KUKA KRL data list: CNC4.dat

&ACCESS RV
DEFDAT CNC4 Public
DECL GLOBAL FRAME gfCNCPoint4[30000]


gfCNCPoint4[1] = {X 250.4410, Y 22.5668, Z -3.9870, A 0.000, B 0.000, C 0.000 }
gfCNCPoint4[2] = {X 251.6873, Y 22.5560, Z -4.3210, A 0.000, B 0.000, C 0.000 }
gfCNCPoint4[3] = {X 252.9774, Y 22.5560, Z -4.6667, A 0.000, B 0.000, C 0.000 }
gfCNCPoint4[4] = {X 257.4115, Y 22.5560, Z -4.6667, A 0.000, B 0.000, C 0.000 }
gfCNCPoint4[5] = {X 257.4115, Y 19.7811, Z -4.6667, A 0.000, B 0.000, C 0.000 }
gfCNCPoint4[6] = {X 251.5292, Y 19.7811, Z -4.6667, A 0.000, B 0.000, C 0.000 }
gfCNCPoint4[7] = {X 250.8345, Y 19.7919, Z -4.6667, A 0.000, B 0.000, C 0.000 }
gfCNCPoint4[8] = {X 249.8296, Y 19.8652, Z -4.6667, A 0.000, B 0.000, C 0.000 }
gfCNCPoint4[9] = {X 248.8453, Y 20.0800, Z -4.6667, A 0.000, B 0.000, C 0.000 }
gfCNCPoint4[10] = {X 248.7005, Y 20.1571, Z -4.6667, A 0.000, B 0.000, C 0.000 }
gfCNCPoint4[11] = {X 248.6143, Y 20.2967, Z -4.6667, A 0.000, B 0.000, C 0.000 }
gfCNCPoint4[12] = {X 248.4764, Y 20.9719, Z -4.6667, A 0.000, B 0.000, C 0.000 }
gfCNCPoint4[13] = {X 248.4575, Y 21.6608, Z -4.6667, A 0.000, B 0.000, C 0.000 }
gfCNCPoint4[14] = {X 248.5584, Y 22.3425, Z -4.6667, A 0.000, B 0.000, C 0.000 }
gfCNCPoint4[15] = {X 248.8771, Y 22.4203, Z -4.6667, A 0.000, B 0.000, C 0.000 }
gfCNCPoint4[16] = {X 249.2022, Y 22.4644, Z -4.6667, A 0.000, B 0.000, C 0.000 }
gfCNCPoint4[17] = {X 250.4437, Y 22.5386, Z -4.6667, A 0.000, B 0.000, C 0.000 }
gfCNCPoint4[18] = {X 251.6873, Y 22.5560, Z -4.6667, A 0.000, B 0.000, C 0.000 }
gfCNCPoint4[19] = {X 252.9774, Y 22.5560, Z -4.6667, A 0.000, B 0.000, C 0.000 }
gfCNCPoint4[20] = {X 248.9926, Y 22.2874, Z -4.6667, A 0.000, B 0.000, C 0.000 }
gfCNCPoint4[21] = {X 252.9774, Y 22.6360, Z -4.6667, A 0.000, B 0.000, C 0.000 }
gfCNCPoint4[22] = {X 257.4915, Y 22.6360, Z -4.6667, A 0.000, B 0.000, C 0.000 }
gfCNCPoint4[23] = {X 257.4915, Y 19.7011, Z -4.6667, A 0.000, B 0.000, C 0.000 }
gfCNCPoint4[24] = {X 251.5286, Y 19.7011, Z -4.6667, A 0.000, B 0.000, C 0.000 }
gfCNCPoint4[25] = {X 250.8365, Y 19.7119, Z -4.6667, A 0.000, B 0.000, C 0.000 }
gfCNCPoint4[26] = {X 249.8259, Y 19.7853, Z -4.6667, A 0.000, B 0.000, C 0.000 }
gfCNCPoint4[27] = {X 248.8356, Y 20.0002, Z -4.6667, A 0.000, B 0.000, C 0.000 }
gfCNCPoint4[28] = {X 248.6488, Y 20.0958, Z -4.6667, A 0.000, B 0.000, C 0.000 }
gfCNCPoint4[29] = {X 248.5376, Y 20.2739, Z -4.6667, A 0.000, B 0.000, C 0.000 }
gfCNCPoint4[30] = {X 248.3952, Y 20.9779, Z -4.6667, A 0.000, B 0.000, C 0.000 }
gfCNCPoint4[31] = {X 248.3796, Y 21.6960, Z -4.6667, A 0.000, B 0.000, C 0.000 }
gfCNCPoint4[32] = {X 248.4915, Y 22.4056, Z -4.6667, A 0.000, B 0.000, C 0.000 }
gfCNCPoint4[33] = {X 248.8397, Y 22.4946, Z -4.6667, A 0.000, B 0.000, C 0.000 }
gfCNCPoint4[34] = {X 249.1956, Y 22.5442, Z -4.6667, A 0.000, B 0.000, C 0.000 }
gfCNCPoint4[35] = {X 250.4397, Y 22.6185, Z -4.6667, A 0.000, B 0.000, C 0.000 }
gfCNCPoint4[36] = {X 251.6859, Y 22.6360, Z -4.6667, A 0.000, B 0.000, C 0.000 }
gfCNCPoint4[37] = {X 252.9774, Y 22.6360, Z -4.6667, A 0.000, B 0.000, C 0.000 }
gfCNCPoint4[38] = {X 256.9621, Y 22.2874, Z -4.6667, A 0.000, B 0.000, C 0.000 }
gfCNCPoint4[39] = {X 248.9926, Y 22.3674, Z -4.6667, A 0.000, B 0.000, C 0.000 }
gfCNCPoint4[40] = {X 252.9774, Y 22.7160, Z -4.6667, A 0.000, B 0.000, C 0.000 }
gfCNCPoint4[41] = {X 257.5715, Y 22.7160, Z -4.6667, A 0.000, B 0.000, C 0.000 }
gfCNCPoint4[42] = {X 257.5715, Y 19.6211, Z -4.6667, A 0.000, B 0.000, C 0.000 }
gfCNCPoint4[43] = {X 251.5280, Y 19.6211, Z -4.6667, A 0.000, B 0.000, C 0.000 }
gfCNCPoint4[44] = {X 250.8358, Y 19.6319, Z -4.6667, A 0.000, B 0.000, C 0.000 }
gfCNCPoint4[45] = {X 249.8156, Y 19.7059, Z -4.6667, A 0.000, B 0.000, C 0.000 }
gfCNCPoint4[46] = {X 248.8160, Y 19.9226, Z -4.6667, A 0.000, B 0.000, C 0.000 }
gfCNCPoint4[47] = {X 248.5934, Y 20.0381, Z -4.6667, A 0.000, B 0.000, C 0.000 }
gfCNCPoint4[48] = {X 248.4609, Y 20.2511, Z -4.6667, A 0.000, B 0.000, C 0.000 }
gfCNCPoint4[49] = {X 248.3140, Y 20.9838, Z -4.6667, A 0.000, B 0.000, C 0.000 }
gfCNCPoint4[50] = {X 248.3019, Y 21.7310, Z -4.6667, A 0.000, B 0.000, C 0.000 }
gfCNCPoint4[51] = {X 248.4249, Y 22.4681, Z -4.6667, A 0.000, B 0.000, C 0.000 }
gfCNCPoint4[52] = {X 248.8023, Y 22.5687, Z -4.6667, A 0.000, B 0.000, C 0.000 }
gfCNCPoint4[53] = {X 249.1890, Y 22.6239, Z -4.6667, A 0.000, B 0.000, C 0.000 }
gfCNCPoint4[54] = {X 250.4366, Y 22.6984, Z -4.6667, A 0.000, B 0.000, C 0.000 }
gfCNCPoint4[55] = {X 251.6863, Y 22.7160, Z -4.6667, A 0.000, B 0.000, C 0.000 }
gfCNCPoint4[56] = {X 252.9774, Y 22.7160, Z -4.6667, A 0.000, B 0.000, C 0.000 }
gfCNCPoint4[57] = {X 256.9621, Y 22.3674, Z -4.6667, A 0.000, B 0.000, C 0.000 }
gfCNCPoint4[58] = {X 248.9926, Y 22.4474, Z -4.6667, A 0.000, B 0.000, C 0.000 }
gfCNCPoint4[59] = {X 252.9774, Y 22.7960, Z -4.6667, A 0.000, B 0.000, C 0.000 }
gfCNCPoint4[60] = {X 257.6515, Y 22.7960, Z -4.6667, A 0.000, B 0.000, C 0.000 }
gfCNCPoint4[61] = {X 257.6515, Y 19.5411, Z -4.6667, A 0.000, B 0.000, C 0.000 }
gfCNCPoint4[62] = {X 251.5274, Y 19.5411, Z -4.6667, A 0.000, B 0.000, C 0.000 }
gfCNCPoint4[63] = {X 250.8351, Y 19.5519, Z -4.6667, A 0.000, B 0.000, C 0.000 }
gfCNCPoint4[64] = {X 249.8053, Y 19.6266, Z -4.6667, A 0.000, B 0.000, C 0.000 }
gfCNCPoint4[65] = {X 248.7962, Y 19.8450, Z -4.6667, A 0.000, B 0.000, C 0.000 }
gfCNCPoint4[66] = {X 248.5379, Y 19.9805, Z -4.6667, A 0.000, B 0.000, C 0.000 }
gfCNCPoint4[67] = {X 248.3842, Y 20.2283, Z -4.6667, A 0.000, B 0.000, C 0.000 }
gfCNCPoint4[68] = {X 248.2330, Y 20.9896, Z -4.6667, A 0.000, B 0.000, C 0.000 }
gfCNCPoint4[69] = {X 248.2244, Y 21.7657, Z -4.6667, A 0.000, B 0.000, C 0.000 }
gfCNCPoint4[70] = {X 248.3587, Y 22.5302, Z -4.6667, A 0.000, B 0.000, C 0.000 }
gfCNCPoint4[71] = {X 248.7651, Y 22.6427, Z -4.6667, A 0.000, B 0.000, C 0.000 }
gfCNCPoint4[72] = {X 249.1825, Y 22.7036, Z -4.6667, A 0.000, B 0.000, C 0.000 }
gfCNCPoint4[73] = {X 250.4335, Y 22.7784, Z -4.6667, A 0.000, B 0.000, C 0.000 }
gfCNCPoint4[74] = {X 251.6866, Y 22.7960, Z -4.6667, A 0.000, B 0.000, C 0.000 }
gfCNCPoint4[75] = {X 252.9774, Y 22.7960, Z -4.6667, A 0.000, B 0.000, C 0.000 }
gfCNCPoint4[76] = {X 256.9621, Y 22.4474, Z -4.6667, A 0.000, B 0.000, C 0.000 }
gfCNCPoint4[77] = {X 248.9926, Y 22.5274, Z -4.6667, A 0.000, B 0.000, C 0.000 }
gfCNCPoint4[78] = {X 252.9774, Y 22.8760, Z -4.6667, A 0.000, B 0.000, C 0.000 }
gfCNCPoint4[79] = {X 257.7315, Y 22.8760, Z -4.6667, A 0.000, B 0.000, C 0.000 }
gfCNCPoint4[80] = {X 257.7315, Y 19.4611, Z -4.6667, A 0.000, B 0.000, C 0.000 }
gfCNCPoint4[81] = {X 251.5267, Y 19.4611, Z -4.6667, A 0.000, B 0.000, C 0.000 }
gfCNCPoint4[82] = {X 250.8343, Y 19.4719, Z -4.6667, A 0.000, B 0.000, C 0.000 }
gfCNCPoint4[83] = {X 249.7949, Y 19.5472, Z -4.6667, A 0.000, B 0.000, C 0.000 }
gfCNCPoint4[84] = {X 248.7763, Y 19.7675, Z -4.6667, A 0.000, B 0.000, C 0.000 }
gfCNCPoint4[85] = {X 248.4824, Y 19.9229, Z -4.6667, A 0.000, B 0.000, C 0.000 }
gfCNCPoint4[86] = {X 248.3075, Y 20.2056, Z -4.6667, A 0.000, B 0.000, C 0.000 }
gfCNCPoint4[87] = {X 248.1526, Y 20.9889, Z -4.6667, A 0.000, B 0.000, C 0.000 }
gfCNCPoint4[88] = {X 248.1459, Y 21.7874, Z -4.6667, A 0.000, B 0.000, C 0.000 }
gfCNCPoint4[89] = {X 248.2876, Y 22.5732, Z -4.6667, A 0.000, B 0.000, C 0.000 }
gfCNCPoint4[90] = {X 248.3062, Y 22.5966, Z -4.6667, A 0.000, B 0.000, C 0.000 }
gfCNCPoint4[91] = {X 248.3326, Y 22.6058, Z -4.6667, A 0.000, B 0.000, C 0.000 }
gfCNCPoint4[92] = {X 248.7487, Y 22.7210, Z -4.6667, A 0.000, B 0.000, C 0.000 }
gfCNCPoint4[93] = {X 249.1759, Y 22.7833, Z -4.6667, A 0.000, B 0.000, C 0.000 }
gfCNCPoint4[94] = {X 250.4304, Y 22.8583, Z -4.6667, A 0.000, B 0.000, C 0.000 }
gfCNCPoint4[95] = {X 251.6870, Y 22.8760, Z -4.6667, A 0.000, B 0.000, C 0.000 }
gfCNCPoint4[96] = {X 252.9774, Y 22.8760, Z -4.6667, A 0.000, B 0.000, C 0.000 }
gfCNCPoint4[97] = {X 256.9621, Y 22.5274, Z -4.6667, A 0.000, B 0.000, C 0.000 }
gfCNCPoint4[98] = {X 248.9926, Y 22.6074, Z -4.6667, A 0.000, B 0.000, C 0.000 }
gfCNCPoint4[99] = {X 252.9774, Y 22.9560, Z -4.6667, A 0.000, B 0.000, C 0.000 }
gfCNCPoint4[100] = {X 257.8115, Y 22.9560, Z -4.6667, A 0.000, B 0.000, C 0.000 }
gfCNCPoint4[101] = {X 257.8115, Y 19.3811, Z -4.6667, A 0.000, B 0.000, C 0.000 }
gfCNCPoint4[102] = {X 251.5261, Y 19.3811, Z -4.6667, A 0.000, B 0.000, C 0.000 }
gfCNCPoint4[103] = {X 250.8336, Y 19.3919, Z -4.6667, A 0.000, B 0.000, C 0.000 }
gfCNCPoint4[104] = {X 249.7844, Y 19.4679, Z -4.6667, A 0.000, B 0.000, C 0.000 }
gfCNCPoint4[105] = {X 248.7562, Y 19.6901, Z -4.6667, A 0.000, B 0.000, C 0.000 }
gfCNCPoint4[106] = {X 248.4268, Y 19.8653, Z -4.6667, A 0.000, B 0.000, C 0.000 }
gfCNCPoint4[107] = {X 248.2308, Y 20.1828, Z -4.6667, A 0.000, B 0.000, C 0.000 }
gfCNCPoint4[108] = {X 248.0725, Y 20.9862, Z -4.6667, A 0.000, B 0.000, C 0.000 }
gfCNCPoint4[109] = {X 248.0671, Y 21.8050, Z -4.6667, A 0.000, B 0.000, C 0.000 }
gfCNCPoint4[110] = {X 248.2149, Y 22.6104, Z -4.6667, A 0.000, B 0.000, C 0.000 }
gfCNCPoint4[111] = {X 248.2579, Y 22.6642, Z -4.6667, A 0.000, B 0.000, C 0.000 }
gfCNCPoint4[112] = {X 248.7070, Y 22.7939, Z -4.6667, A 0.000, B 0.000, C 0.000 }
gfCNCPoint4[113] = {X 249.1693, Y 22.8631, Z -4.6667, A 0.000, B 0.000, C 0.000 }
gfCNCPoint4[114] = {X 250.4273, Y 22.9382, Z -4.6667, A 0.000, B 0.000, C 0.000 }
gfCNCPoint4[115] = {X 251.6873, Y 22.9560, Z -4.6667, A 0.000, B 0.000, C 0.000 }
gfCNCPoint4[116] = {X 252.9774, Y 22.9560, Z -4.6667, A 0.000, B 0.000, C 0.000 }
gfCNCPoint4[117] = {X 256.9621, Y 22.6074, Z -4.6667, A 0.000, B 0.000, C 0.000 }
gfCNCPoint4[118] = {X 256.9621, Y 22.6074, Z -1.6667, A 0.000, B 0.000, C 0.000 }
gfCNCPoint4[119] = {X 256.9621, Y 22.6074, Z 11.0000, A 0.000, B 0.000, C 0.000 }
gfCNCPoint4[120] = {X 188.4967, Y 19.4668, Z 11.0000, A 0.000, B 0.000, C 0.000 }
gfCNCPoint4[121] = {X 188.4967, Y 19.4668, Z -0.8333, A 0.000, B 0.000, C 0.000 }
gfCNCPoint4[122] = {X 188.3884, Y 19.4285, Z -0.8641, A 0.000, B 0.000, C 0.000 }
gfCNCPoint4[123] = {X 187.7714, Y 19.3599, Z -1.0305, A 0.000, B 0.000, C 0.000 }
gfCNCPoint4[124] = {X 186.9109, Y 19.2599, Z -1.2626, A 0.000, B 0.000, C 0.000 }
gfCNCPoint4[125] = {X 184.5930, Y 19.3674, Z -1.8843, A 0.000, B 0.000, C 0.000 }
gfCNCPoint4[126] = {X 183.7426, Y 19.5472, Z -2.1172, A 0.000, B 0.000, C 0.000 }
gfCNCPoint4[127] = {X 183.0434, Y 19.6897, Z -2.3084, A 0.000, B 0.000, C 0.000 }
gfCNCPoint4[128] = {X 182.0228, Y 20.0611, Z -2.5995, A 0.000, B 0.000, C 0.000 }
gfCNCPoint4[129] = {X 181.3955, Y 20.4013, Z -2.7907, A 0.000, B 0.000, C 0.000 }
gfCNCPoint4[130] = {X 181.3396, Y 20.9130, Z -2.9286, A 0.000, B 0.000, C 0.000 }
gfCNCPoint4[131] = {X 180.8648, Y 22.1264, Z -3.2777, A 0.000, B 0.000, C 0.000 }
gfCNCPoint4[132] = {X 180.5586, Y 22.5402, Z -3.4156, A 0.000, B 0.000, C 0.000 }
gfCNCPoint4[133] = {X 182.2913, Y 22.3342, Z -3.8832, A 0.000, B 0.000, C 0.000 }
gfCNCPoint4[134] = {X 182.5945, Y 22.3096, Z -3.9647, A 0.000, B 0.000, C 0.000 }
gfCNCPoint4[135] = {X 184.3413, Y 22.2335, Z -4.4332, A 0.000, B 0.000, C 0.000 }
gfCNCPoint4[136] = {X 184.7767, Y 22.2184, Z -4.5499, A 0.000, B 0.000, C 0.000 }
gfCNCPoint4[137] = {X 185.2120, Y 22.2000, Z -4.6667, A 0.000, B 0.000, C 0.000 }
gfCNCPoint4[138] = {X 187.5425, Y 22.0775, Z -4.6667, A 0.000, B 0.000, C 0.000 }
gfCNCPoint4[139] = {X 189.8699, Y 21.9072, Z -4.6667, A 0.000, B 0.000, C 0.000 }
gfCNCPoint4[140] = {X 190.4714, Y 21.8310, Z -4.6667, A 0.000, B 0.000, C 0.000 }
gfCNCPoint4[141] = {X 191.0586, Y 21.6797, Z -4.6667, A 0.000, B 0.000, C 0.000 }
gfCNCPoint4[142] = {X 191.0683, Y 21.1639, Z -4.6667, A 0.000, B 0.000, C 0.000 }
gfCNCPoint4[143] = {X 190.8726, Y 20.6866, Z -4.6667, A 0.000, B 0.000, C 0.000 }
gfCNCPoint4[144] = {X 190.5035, Y 20.3261, Z -4.6667, A 0.000, B 0.000, C 0.000 }
gfCNCPoint4[145] = {X 189.6459, Y 19.8654, Z -4.6667, A 0.000, B 0.000, C 0.000 }
gfCNCPoint4[146] = {X 188.7280, Y 19.5408, Z -4.6667, A 0.000, B 0.000, C 0.000 }
gfCNCPoint4[147] = {X 187.7714, Y 19.3599, Z -4.6667, A 0.000, B 0.000, C 0.000 }
gfCNCPoint4[148] = {X 186.4243, Y 19.2768, Z -4.6667, A 0.000, B 0.000, C 0.000 }
gfCNCPoint4[149] = {X 185.0761, Y 19.3395, Z -4.6667, A 0.000, B 0.000, C 0.000 }
gfCNCPoint4[150] = {X 183.7426, Y 19.5472, Z -4.6667, A 0.000, B 0.000, C 0.000 }
gfCNCPoint4[151] = {X 182.5374, Y 19.8873, Z -4.6667, A 0.000, B 0.000, C 0.000 }
gfCNCPoint4[152] = {X 181.3955, Y 20.4013, Z -4.6667, A 0.000, B 0.000, C 0.000 }
gfCNCPoint4[153] = {X 181.2441, Y 21.1599, Z -4.6667, A 0.000, B 0.000, C 0.000 }
gfCNCPoint4[154] = {X 180.9623, Y 21.8803, Z -4.6667, A 0.000, B 0.000, C 0.000 }
gfCNCPoint4[155] = {X 180.5586, Y 22.5402, Z -4.6667, A 0.000, B 0.000, C 0.000 }
gfCNCPoint4[156] = {X 182.4471, Y 22.3514, Z -4.6667, A 0.000, B 0.000, C 0.000 }
gfCNCPoint4[157] = {X 184.3413, Y 22.2335, Z -4.6667, A 0.000, B 0.000, C 0.000 }
gfCNCPoint4[158] = {X 184.7767, Y 22.2176, Z -4.6667, A 0.000, B 0.000, C 0.000 }
gfCNCPoint4[159] = {X 185.2120, Y 22.2000, Z -4.6667, A 0.000, B 0.000, C 0.000 }
gfCNCPoint4[160] = {X 181.2195, Y 22.1000, Z -4.6667, A 0.000, B 0.000, C 0.000 }
gfCNCPoint4[161] = {X 185.2154, Y 22.2799, Z -4.6667, A 0.000, B 0.000, C 0.000 }
gfCNCPoint4[162] = {X 187.5451, Y 22.1574, Z -4.6667, A 0.000, B 0.000, C 0.000 }
gfCNCPoint4[163] = {X 189.8717, Y 21.9873, Z -4.6667, A 0.000, B 0.000, C 0.000 }
gfCNCPoint4[164] = {X 190.5068, Y 21.9056, Z -4.6667, A 0.000, B 0.000, C 0.000 }
gfCNCPoint4[165] = {X 191.1258, Y 21.7417, Z -4.6667, A 0.000, B 0.000, C 0.000 }
gfCNCPoint4[166] = {X 191.1522, Y 21.1791, Z -4.6667, A 0.000, B 0.000, C 0.000 }
gfCNCPoint4[167] = {X 190.9473, Y 20.6545, Z -4.6667, A 0.000, B 0.000, C 0.000 }
gfCNCPoint4[168] = {X 190.5466, Y 20.2588, Z -4.6667, A 0.000, B 0.000, C 0.000 }
gfCNCPoint4[169] = {X 189.6789, Y 19.7925, Z -4.6667, A 0.000, B 0.000, C 0.000 }
gfCNCPoint4[170] = {X 188.7502, Y 19.4639, Z -4.6667, A 0.000, B 0.000, C 0.000 }
gfCNCPoint4[171] = {X 187.7823, Y 19.2806, Z -4.6667, A 0.000, B 0.000, C 0.000 }
gfCNCPoint4[172] = {X 186.4270, Y 19.1968, Z -4.6667, A 0.000, B 0.000, C 0.000 }
gfCNCPoint4[173] = {X 185.0706, Y 19.2596, Z -4.6667, A 0.000, B 0.000, C 0.000 }
gfCNCPoint4[174] = {X 183.7289, Y 19.4683, Z -4.6667, A 0.000, B 0.000, C 0.000 }
gfCNCPoint4[175] = {X 182.4920, Y 19.8187, Z -4.6667, A 0.000, B 0.000, C 0.000 }
gfCNCPoint4[176] = {X 181.3216, Y 20.3505, Z -4.6667, A 0.000, B 0.000, C 0.000 }
gfCNCPoint4[177] = {X 181.1594, Y 21.1706, Z -4.6667, A 0.000, B 0.000, C 0.000 }
gfCNCPoint4[178] = {X 180.8424, Y 21.9441, Z -4.6667, A 0.000, B 0.000, C 0.000 }
gfCNCPoint4[179] = {X 180.3824, Y 22.6420, Z -4.6667, A 0.000, B 0.000, C 0.000 }
gfCNCPoint4[180] = {X 182.3593, Y 22.4389, Z -4.6667, A 0.000, B 0.000, C 0.000 }
gfCNCPoint4[181] = {X 184.3427, Y 22.3135, Z -4.6667, A 0.000, B 0.000, C 0.000 }
gfCNCPoint4[182] = {X 184.7791, Y 22.2975, Z -4.6667, A 0.000, B 0.000, C 0.000 }
gfCNCPoint4[183] = {X 185.2154, Y 22.2799, Z -4.6667, A 0.000, B 0.000, C 0.000 }
gfCNCPoint4[184] = {X 189.1819, Y 21.7632, Z -4.6667, A 0.000, B 0.000, C 0.000 }
gfCNCPoint4[185] = {X 181.2228, Y 22.1799, Z -4.6667, A 0.000, B 0.000, C 0.000 }
gfCNCPoint4[186] = {X 185.2188, Y 22.3598, Z -4.6667, A 0.000, B 0.000, C 0.000 }
gfCNCPoint4[187] = {X 187.5497, Y 22.2373, Z -4.6667, A 0.000, B 0.000, C 0.000 }
gfCNCPoint4[188] = {X 189.8775, Y 22.0671, Z -4.6667, A 0.000, B 0.000, C 0.000 }
gfCNCPoint4[189] = {X 190.5434, Y 21.9799, Z -4.6667, A 0.000, B 0.000, C 0.000 }
gfCNCPoint4[190] = {X 191.1915, Y 21.8038, Z -4.6667, A 0.000, B 0.000, C 0.000 }
gfCNCPoint4[191] = {X 191.2492, Y 21.3479, Z -4.6667, A 0.000, B 0.000, C 0.000 }
gfCNCPoint4[192] = {X 191.1596, Y 20.8972, Z -4.6667, A 0.000, B 0.000, C 0.000 }
gfCNCPoint4[193] = {X 190.9320, Y 20.4980, Z -4.6667, A 0.000, B 0.000, C 0.000 }
gfCNCPoint4[194] = {X 190.5898, Y 20.1914, Z -4.6667, A 0.000, B 0.000, C 0.000 }
gfCNCPoint4[195] = {X 189.7112, Y 19.7193, Z -4.6667, A 0.000, B 0.000, C 0.000 }
gfCNCPoint4[196] = {X 188.7710, Y 19.3866, Z -4.6667, A 0.000, B 0.000, C 0.000 }
gfCNCPoint4[197] = {X 187.7911, Y 19.2011, Z -4.6667, A 0.000, B 0.000, C 0.000 }
gfCNCPoint4[198] = {X 186.4273, Y 19.1168, Z -4.6667, A 0.000, B 0.000, C 0.000 }
gfCNCPoint4[199] = {X 185.0625, Y 19.1800, Z -4.6667, A 0.000, B 0.000, C 0.000 }
gfCNCPoint4[200] = {X 183.7123, Y 19.3901, Z -4.6667, A 0.000, B 0.000, C 0.000 }
gfCNCPoint4[201] = {X 182.4464, Y 19.7502, Z -4.6667, A 0.000, B 0.000, C 0.000 }
gfCNCPoint4[202] = {X 181.2499, Y 20.2987, Z -4.6667, A 0.000, B 0.000, C 0.000 }
gfCNCPoint4[203] = {X 181.2398, Y 20.3526, Z -4.6667, A 0.000, B 0.000, C 0.000 }
gfCNCPoint4[204] = {X 181.0600, Y 21.2185, Z -4.6667, A 0.000, B 0.000, C 0.000 }
gfCNCPoint4[205] = {X 180.7045, Y 22.0284, Z -4.6667, A 0.000, B 0.000, C 0.000 }
gfCNCPoint4[206] = {X 180.1887, Y 22.7468, Z -4.6667, A 0.000, B 0.000, C 0.000 }
gfCNCPoint4[207] = {X 182.2636, Y 22.5272, Z -4.6667, A 0.000, B 0.000, C 0.000 }
gfCNCPoint4[208] = {X 184.3458, Y 22.3934, Z -4.6667, A 0.000, B 0.000, C 0.000 }
gfCNCPoint4[209] = {X 184.7823, Y 22.3775, Z -4.6667, A 0.000, B 0.000, C 0.000 }
gfCNCPoint4[210] = {X 185.2188, Y 22.3598, Z -4.6667, A 0.000, B 0.000, C 0.000 }
gfCNCPoint4[211] = {X 189.1853, Y 21.8431, Z -4.6667, A 0.000, B 0.000, C 0.000 }
gfCNCPoint4[212] = {X 181.2262, Y 22.2599, Z -4.6667, A 0.000, B 0.000, C 0.000 }
gfCNCPoint4[213] = {X 185.2222, Y 22.4398, Z -4.6667, A 0.000, B 0.000, C 0.000 }
gfCNCPoint4[214] = {X 187.5543, Y 22.3172, Z -4.6667, A 0.000, B 0.000, C 0.000 }
gfCNCPoint4[215] = {X 189.8834, Y 22.1469, Z -4.6667, A 0.000, B 0.000, C 0.000 }
gfCNCPoint4[216] = {X 190.5795, Y 22.0543, Z -4.6667, A 0.000, B 0.000, C 0.000 }
gfCNCPoint4[217] = {X 191.2560, Y 21.8660, Z -4.6667, A 0.000, B 0.000, C 0.000 }
gfCNCPoint4[218] = {X 191.3299, Y 21.3762, Z -4.6667, A 0.000, B 0.000, C 0.000 }
gfCNCPoint4[219] = {X 191.2417, Y 20.8887, Z -4.6667, A 0.000, B 0.000, C 0.000 }
gfCNCPoint4[220] = {X 191.0007, Y 20.4558, Z -4.6667, A 0.000, B 0.000, C 0.000 }
gfCNCPoint4[221] = {X 190.6329, Y 20.1240, Z -4.6667, A 0.000, B 0.000, C 0.000 }
gfCNCPoint4[222] = {X 189.7436, Y 19.6462, Z -4.6667, A 0.000, B 0.000, C 0.000 }
gfCNCPoint4[223] = {X 188.7919, Y 19.3094, Z -4.6667, A 0.000, B 0.000, C 0.000 }
gfCNCPoint4[224] = {X 187.7999, Y 19.1216, Z -4.6667, A 0.000, B 0.000, C 0.000 }
gfCNCPoint4[225] = {X 186.4277, Y 19.0368, Z -4.6667, A 0.000, B 0.000, C 0.000 }
gfCNCPoint4[226] = {X 185.0543, Y 19.1005, Z -4.6667, A 0.000, B 0.000, C 0.000 }
gfCNCPoint4[227] = {X 183.6958, Y 19.3118, Z -4.6667, A 0.000, B 0.000, C 0.000 }
gfCNCPoint4[228] = {X 182.4008, Y 19.6818, Z -4.6667, A 0.000, B 0.000, C 0.000 }
gfCNCPoint4[229] = {X 181.1783, Y 20.2470, Z -4.6667, A 0.000, B 0.000, C 0.000 }
gfCNCPoint4[230] = {X 181.1605, Y 20.3411, Z -4.6667, A 0.000, B 0.000, C 0.000 }
gfCNCPoint4[231] = {X 180.9651, Y 21.2476, Z -4.6667, A 0.000, B 0.000, C 0.000 }
gfCNCPoint4[232] = {X 180.5737, Y 22.0883, Z -4.6667, A 0.000, B 0.000, C 0.000 }
gfCNCPoint4[233] = {X 180.0058, Y 22.8213, Z -4.6667, A 0.000, B 0.000, C 0.000 }
gfCNCPoint4[234] = {X 180.1926, Y 22.8270, Z -4.6667, A 0.000, B 0.000, C 0.000 }
gfCNCPoint4[235] = {X 182.2671, Y 22.6072, Z -4.6667, A 0.000, B 0.000, C 0.000 }
gfCNCPoint4[236] = {X 184.3489, Y 22.4734, Z -4.6667, A 0.000, B 0.000, C 0.000 }
gfCNCPoint4[237] = {X 184.7856, Y 22.4574, Z -4.6667, A 0.000, B 0.000, C 0.000 }
gfCNCPoint4[238] = {X 185.2222, Y 22.4398, Z -4.6667, A 0.000, B 0.000, C 0.000 }
gfCNCPoint4[239] = {X 189.1887, Y 21.9231, Z -4.6667, A 0.000, B 0.000, C 0.000 }
gfCNCPoint4[240] = {X 181.2296, Y 22.3398, Z -4.6667, A 0.000, B 0.000, C 0.000 }
gfCNCPoint4[241] = {X 185.2256, Y 22.5197, Z -4.6667, A 0.000, B 0.000, C 0.000 }
gfCNCPoint4[242] = {X 187.5589, Y 22.3971, Z -4.6667, A 0.000, B 0.000, C 0.000 }
gfCNCPoint4[243] = {X 189.8892, Y 22.2267, Z -4.6667, A 0.000, B 0.000, C 0.000 }
gfCNCPoint4[244] = {X 190.6150, Y 22.1286, Z -4.6667, A 0.000, B 0.000, C 0.000 }
gfCNCPoint4[245] = {X 191.3193, Y 21.9282, Z -4.6667, A 0.000, B 0.000, C 0.000 }
gfCNCPoint4[246] = {X 191.4101, Y 21.4047, Z -4.6667, A 0.000, B 0.000, C 0.000 }
gfCNCPoint4[247] = {X 191.3236, Y 20.8804, Z -4.6667, A 0.000, B 0.000, C 0.000 }
gfCNCPoint4[248] = {X 191.0695, Y 20.4138, Z -4.6667, A 0.000, B 0.000, C 0.000 }
gfCNCPoint4[249] = {X 190.6760, Y 20.0566, Z -4.6667, A 0.000, B 0.000, C 0.000 }
gfCNCPoint4[250] = {X 189.7760, Y 19.5730, Z -4.6667, A 0.000, B 0.000, C 0.000 }
gfCNCPoint4[251] = {X 188.8127, Y 19.2322, Z -4.6667, A 0.000, B 0.000, C 0.000 }
gfCNCPoint4[252] = {X 187.8088, Y 19.0421, Z -4.6667, A 0.000, B 0.000, C 0.000 }
gfCNCPoint4[253] = {X 186.4280, Y 18.9568, Z -4.6667, A 0.000, B 0.000, C 0.000 }
gfCNCPoint4[254] = {X 185.0462, Y 19.0209, Z -4.6667, A 0.000, B 0.000, C 0.000 }
gfCNCPoint4[255] = {X 183.6792, Y 19.2335, Z -4.6667, A 0.000, B 0.000, C 0.000 }
gfCNCPoint4[256] = {X 182.3551, Y 19.6135, Z -4.6667, A 0.000, B 0.000, C 0.000 }
gfCNCPoint4[257] = {X 181.1066, Y 20.1956, Z -4.6667, A 0.000, B 0.000, C 0.000 }
gfCNCPoint4[258] = {X 181.0813, Y 20.3297, Z -4.6667, A 0.000, B 0.000, C 0.000 }
gfCNCPoint4[259] = {X 180.8699, Y 21.2784, Z -4.6667, A 0.000, B 0.000, C 0.000 }
gfCNCPoint4[260] = {X 180.4401, Y 22.1503, Z -4.6667, A 0.000, B 0.000, C 0.000 }
gfCNCPoint4[261] = {X 179.8162, Y 22.8957, Z -4.6667, A 0.000, B 0.000, C 0.000 }
gfCNCPoint4[262] = {X 180.1964, Y 22.9071, Z -4.6667, A 0.000, B 0.000, C 0.000 }
gfCNCPoint4[263] = {X 182.2706, Y 22.6872, Z -4.6667, A 0.000, B 0.000, C 0.000 }
gfCNCPoint4[264] = {X 184.3521, Y 22.5533, Z -4.6667, A 0.000, B 0.000, C 0.000 }
gfCNCPoint4[265] = {X 184.7888, Y 22.5373, Z -4.6667, A 0.000, B 0.000, C 0.000 }
gfCNCPoint4[266] = {X 185.2256, Y 22.5197, Z -4.6667, A 0.000, B 0.000, C 0.000 }
gfCNCPoint4[267] = {X 189.1920, Y 22.0030, Z -4.6667, A 0.000, B 0.000, C 0.000 }
gfCNCPoint4[268] = {X 185.1539, Y 22.6028, Z -4.6667, A 0.000, B 0.000, C 0.000 }
gfCNCPoint4[269] = {X 185.2289, Y 22.5996, Z -4.6667, A 0.000, B 0.000, C 0.000 }
gfCNCPoint4[270] = {X 187.5635, Y 22.4769, Z -4.6667, A 0.000, B 0.000, C 0.000 }
gfCNCPoint4[271] = {X 189.8950, Y 22.3064, Z -4.6667, A 0.000, B 0.000, C 0.000 }
gfCNCPoint4[272] = {X 190.6500, Y 22.2030, Z -4.6667, A 0.000, B 0.000, C 0.000 }
gfCNCPoint4[273] = {X 191.3817, Y 21.9905, Z -4.6667, A 0.000, B 0.000, C 0.000 }
gfCNCPoint4[274] = {X 191.4897, Y 21.4335, Z -4.6667, A 0.000, B 0.000, C 0.000 }
gfCNCPoint4[275] = {X 191.4053, Y 20.8724, Z -4.6667, A 0.000, B 0.000, C 0.000 }
gfCNCPoint4[276] = {X 191.1382, Y 20.3718, Z -4.6667, A 0.000, B 0.000, C 0.000 }
gfCNCPoint4[277] = {X 190.7192, Y 19.9893, Z -4.6667, A 0.000, B 0.000, C 0.000 }
gfCNCPoint4[278] = {X 189.8083, Y 19.4998, Z -4.6667, A 0.000, B 0.000, C 0.000 }
gfCNCPoint4[279] = {X 188.8336, Y 19.1549, Z -4.6667, A 0.000, B 0.000, C 0.000 }
gfCNCPoint4[280] = {X 187.8176, Y 18.9626, Z -4.6667, A 0.000, B 0.000, C 0.000 }
gfCNCPoint4[281] = {X 186.4284, Y 18.8768, Z -4.6667, A 0.000, B 0.000, C 0.000 }
gfCNCPoint4[282] = {X 185.0380, Y 18.9413, Z -4.6667, A 0.000, B 0.000, C 0.000 }
gfCNCPoint4[283] = {X 183.6627, Y 19.1553, Z -4.6667, A 0.000, B 0.000, C 0.000 }
gfCNCPoint4[284] = {X 182.3094, Y 19.5452, Z -4.6667, A 0.000, B 0.000, C 0.000 }
gfCNCPoint4[285] = {X 181.0348, Y 20.1443, Z -4.6667, A 0.000, B 0.000, C 0.000 }
gfCNCPoint4[286] = {X 181.0020, Y 20.3183, Z -4.6667, A 0.000, B 0.000, C 0.000 }
gfCNCPoint4[287] = {X 180.8538, Y 21.0695, Z -4.6667, A 0.000, B 0.000, C 0.000 }
gfCNCPoint4[288] = {X 180.5651, Y 21.7787, Z -4.6667, A 0.000, B 0.000, C 0.000 }
gfCNCPoint4[289] = {X 180.1466, Y 22.4199, Z -4.6667, A 0.000, B 0.000, C 0.000 }
gfCNCPoint4[290] = {X 179.6136, Y 22.9696, Z -4.6667, A 0.000, B 0.000, C 0.000 }
gfCNCPoint4[291] = {X 180.2003, Y 22.9873, Z -4.6667, A 0.000, B 0.000, C 0.000 }
gfCNCPoint4[292] = {X 182.2741, Y 22.7672, Z -4.6667, A 0.000, B 0.000, C 0.000 }
gfCNCPoint4[293] = {X 184.3552, Y 22.6332, Z -4.6667, A 0.000, B 0.000, C 0.000 }
gfCNCPoint4[294] = {X 184.7921, Y 22.6173, Z -4.6667, A 0.000, B 0.000, C 0.000 }
gfCNCPoint4[295] = {X 185.2289, Y 22.5996, Z -4.6667, A 0.000, B 0.000, C 0.000 }
gfCNCPoint4[296] = {X 185.1444, Y 20.6014, Z -4.6667, A 0.000, B 0.000, C 0.000 }
gfCNCPoint4[297] = {X 185.1444, Y 20.6014, Z -1.6667, A 0.000, B 0.000, C 0.000 }
gfCNCPoint4[298] = {X 185.1444, Y 20.6014, Z 11.0000, A 0.000, B 0.000, C 0.000 }
gfCNCPoint4[299] = {X 186.2289, Y 37.9123, Z 11.0000, A 0.000, B 0.000, C 0.000 }
gfCNCPoint4[300] = {X 186.2289, Y 37.9123, Z -0.8333, A 0.000, B 0.000, C 0.000 }
gfCNCPoint4[301] = {X 187.5894, Y 37.8326, Z -1.1985, A 0.000, B 0.000, C 0.000 }
gfCNCPoint4[302] = {X 189.4164, Y 37.3864, Z -1.7024, A 0.000, B 0.000, C 0.000 }
gfCNCPoint4[303] = {X 190.1416, Y 37.0746, Z -1.9139, A 0.000, B 0.000, C 0.000 }
gfCNCPoint4[304] = {X 190.9792, Y 36.7144, Z -2.1583, A 0.000, B 0.000, C 0.000 }
gfCNCPoint4[305] = {X 191.6922, Y 36.3239, Z -2.3761, A 0.000, B 0.000, C 0.000 }
gfCNCPoint4[306] = {X 192.4466, Y 35.8119, Z -2.6204, A 0.000, B 0.000, C 0.000 }
gfCNCPoint4[307] = {X 192.4699, Y 35.2977, Z -2.7583, A 0.000, B 0.000, C 0.000 }
gfCNCPoint4[308] = {X 192.6314, Y 34.6347, Z -2.9411, A 0.000, B 0.000, C 0.000 }
gfCNCPoint4[309] = {X 192.8470, Y 34.1673, Z -3.0791, A 0.000, B 0.000, C 0.000 }
gfCNCPoint4[310] = {X 192.7389, Y 34.1925, Z -3.1088, A 0.000, B 0.000, C 0.000 }
gfCNCPoint4[311] = {X 191.4088, Y 34.4428, Z -3.4715, A 0.000, B 0.000, C 0.000 }
gfCNCPoint4[312] = {X 190.5807, Y 34.5493, Z -3.6952, A 0.000, B 0.000, C 0.000 }
gfCNCPoint4[313] = {X 189.2271, Y 34.6442, Z -4.0588, A 0.000, B 0.000, C 0.000 }
gfCNCPoint4[314] = {X 186.9626, Y 34.7832, Z -4.6667, A 0.000, B 0.000, C 0.000 }
gfCNCPoint4[315] = {X 182.5755, Y 35.0526, Z -4.6667, A 0.000, B 0.000, C 0.000 }
gfCNCPoint4[316] = {X 181.8173, Y 35.1400, Z -4.6667, A 0.000, B 0.000, C 0.000 }
gfCNCPoint4[317] = {X 181.0728, Y 35.3079, Z -4.6667, A 0.000, B 0.000, C 0.000 }
gfCNCPoint4[318] = {X 181.0647, Y 35.3822, Z -4.6667, A 0.000, B 0.000, C 0.000 }
gfCNCPoint4[319] = {X 181.0648, Y 35.4569, Z -4.6667, A 0.000, B 0.000, C 0.000 }
gfCNCPoint4[320] = {X 181.1576, Y 35.9999, Z -4.6667, A 0.000, B 0.000, C 0.000 }
gfCNCPoint4[321] = {X 181.4147, Y 36.4871, Z -4.6667, A 0.000, B 0.000, C 0.000 }
gfCNCPoint4[322] = {X 181.8107, Y 36.8701, Z -4.6667, A 0.000, B 0.000, C 0.000 }
gfCNCPoint4[323] = {X 182.4284, Y 37.2229, Z -4.6667, A 0.000, B 0.000, C 0.000 }
gfCNCPoint4[324] = {X 183.0887, Y 37.4876, Z -4.6667, A 0.000, B 0.000, C 0.000 }
gfCNCPoint4[325] = {X 184.4948, Y 37.8014, Z -4.6667, A 0.000, B 0.000, C 0.000 }
gfCNCPoint4[326] = {X 185.9308, Y 37.9173, Z -4.6667, A 0.000, B 0.000, C 0.000 }
gfCNCPoint4[327] = {X 187.3690, Y 37.8331, Z -4.6667, A 0.000, B 0.000, C 0.000 }
gfCNCPoint4[328] = {X 188.7817, Y 37.5503, Z -4.6667, A 0.000, B 0.000, C 0.000 }
gfCNCPoint4[329] = {X 190.1416, Y 37.0746, Z -4.6667, A 0.000, B 0.000, C 0.000 }
gfCNCPoint4[330] = {X 191.3242, Y 36.4981, Z -4.6667, A 0.000, B 0.000, C 0.000 }
gfCNCPoint4[331] = {X 192.4466, Y 35.8119, Z -4.6667, A 0.000, B 0.000, C 0.000 }
gfCNCPoint4[332] = {X 192.5670, Y 34.9702, Z -4.6667, A 0.000, B 0.000, C 0.000 }
gfCNCPoint4[333] = {X 192.8470, Y 34.1673, Z -4.6667, A 0.000, B 0.000, C 0.000 }
gfCNCPoint4[334] = {X 192.7389, Y 34.1925, Z -4.6667, A 0.000, B 0.000, C 0.000 }
gfCNCPoint4[335] = {X 190.9896, Y 34.4693, Z -4.6667, A 0.000, B 0.000, C 0.000 }
gfCNCPoint4[336] = {X 189.2271, Y 34.6442, Z -4.6667, A 0.000, B 0.000, C 0.000 }
gfCNCPoint4[337] = {X 186.9626, Y 34.7832, Z -4.6667, A 0.000, B 0.000, C 0.000 }
gfCNCPoint4[338] = {X 190.9564, Y 34.8072, Z -4.6667, A 0.000, B 0.000, C 0.000 }
gfCNCPoint4[339] = {X 186.9577, Y 34.7034, Z -4.6667, A 0.000, B 0.000, C 0.000 }
gfCNCPoint4[340] = {X 182.5706, Y 34.9728, Z -4.6667, A 0.000, B 0.000, C 0.000 }
gfCNCPoint4[341] = {X 181.7797, Y 35.0653, Z -4.6667, A 0.000, B 0.000, C 0.000 }
gfCNCPoint4[342] = {X 181.0039, Y 35.2444, Z -4.6667, A 0.000, B 0.000, C 0.000 }
gfCNCPoint4[343] = {X 180.9871, Y 35.3481, Z -4.6667, A 0.000, B 0.000, C 0.000 }
gfCNCPoint4[344] = {X 180.9847, Y 35.4530, Z -4.6667, A 0.000, B 0.000, C 0.000 }
gfCNCPoint4[345] = {X 181.0809, Y 36.0229, Z -4.6667, A 0.000, B 0.000, C 0.000 }
gfCNCPoint4[346] = {X 181.3502, Y 36.5343, Z -4.6667, A 0.000, B 0.000, C 0.000 }
gfCNCPoint4[347] = {X 181.7656, Y 36.9361, Z -4.6667, A 0.000, B 0.000, C 0.000 }
gfCNCPoint4[348] = {X 182.3936, Y 37.2949, Z -4.6667, A 0.000, B 0.000, C 0.000 }
gfCNCPoint4[349] = {X 183.0650, Y 37.5640, Z -4.6667, A 0.000, B 0.000, C 0.000 }
gfCNCPoint4[350] = {X 184.4821, Y 37.8804, Z -4.6667, A 0.000, B 0.000, C 0.000 }
gfCNCPoint4[351] = {X 185.9294, Y 37.9973, Z -4.6667, A 0.000, B 0.000, C 0.000 }
gfCNCPoint4[352] = {X 187.3789, Y 37.9125, Z -4.6667, A 0.000, B 0.000, C 0.000 }
gfCNCPoint4[353] = {X 188.8027, Y 37.6276, Z -4.6667, A 0.000, B 0.000, C 0.000 }
gfCNCPoint4[354] = {X 190.1732, Y 37.1481, Z -4.6667, A 0.000, B 0.000, C 0.000 }
gfCNCPoint4[355] = {X 191.3803, Y 36.5585, Z -4.6667, A 0.000, B 0.000, C 0.000 }
gfCNCPoint4[356] = {X 192.5249, Y 35.8553, Z -4.6667, A 0.000, B 0.000, C 0.000 }
gfCNCPoint4[357] = {X 192.6602, Y 34.9275, Z -4.6667, A 0.000, B 0.000, C 0.000 }
gfCNCPoint4[358] = {X 192.9925, Y 34.0506, Z -4.6667, A 0.000, B 0.000, C 0.000 }
gfCNCPoint4[359] = {X 192.7315, Y 34.1125, Z -4.6667, A 0.000, B 0.000, C 0.000 }
gfCNCPoint4[360] = {X 190.9841, Y 34.3894, Z -4.6667, A 0.000, B 0.000, C 0.000 }
gfCNCPoint4[361] = {X 189.2236, Y 34.5643, Z -4.6667, A 0.000, B 0.000, C 0.000 }
gfCNCPoint4[362] = {X 186.9577, Y 34.7034, Z -4.6667, A 0.000, B 0.000, C 0.000 }
gfCNCPoint4[363] = {X 183.0018, Y 35.2956, Z -4.6667, A 0.000, B 0.000, C 0.000 }
gfCNCPoint4[364] = {X 190.9515, Y 34.7273, Z -4.6667, A 0.000, B 0.000, C 0.000 }
gfCNCPoint4[365] = {X 186.9528, Y 34.6235, Z -4.6667, A 0.000, B 0.000, C 0.000 }
gfCNCPoint4[366] = {X 182.5657, Y 34.8929, Z -4.6667, A 0.000, B 0.000, C 0.000 }
gfCNCPoint4[367] = {X 181.7437, Y 34.9904, Z -4.6667, A 0.000, B 0.000, C 0.000 }
gfCNCPoint4[368] = {X 180.9381, Y 35.1804, Z -4.6667, A 0.000, B 0.000, C 0.000 }
gfCNCPoint4[369] = {X 180.9101, Y 35.3164, Z -4.6667, A 0.000, B 0.000, C 0.000 }
gfCNCPoint4[370] = {X 180.9047, Y 35.4551, Z -4.6667, A 0.000, B 0.000, C 0.000 }
gfCNCPoint4[371] = {X 181.0055, Y 36.0497, Z -4.6667, A 0.000, B 0.000, C 0.000 }
gfCNCPoint4[372] = {X 181.2868, Y 36.5832, Z -4.6667, A 0.000, B 0.000, C 0.000 }
gfCNCPoint4[373] = {X 181.7205, Y 37.0022, Z -4.6667, A 0.000, B 0.000, C 0.000 }
gfCNCPoint4[374] = {X 182.3588, Y 37.3670, Z -4.6667, A 0.000, B 0.000, C 0.000 }
gfCNCPoint4[375] = {X 183.0413, Y 37.6404, Z -4.6667, A 0.000, B 0.000, C 0.000 }
gfCNCPoint4[376] = {X 184.4694, Y 37.9593, Z -4.6667, A 0.000, B 0.000, C 0.000 }
gfCNCPoint4[377] = {X 185.9279, Y 38.0773, Z -4.6667, A 0.000, B 0.000, C 0.000 }
gfCNCPoint4[378] = {X 187.3887, Y 37.9918, Z -4.6667, A 0.000, B 0.000, C 0.000 }
gfCNCPoint4[379] = {X 188.8236, Y 37.7048, Z -4.6667, A 0.000, B 0.000, C 0.000 }
gfCNCPoint4[380] = {X 190.2048, Y 37.2216, Z -4.6667, A 0.000, B 0.000, C 0.000 }
gfCNCPoint4[381] = {X 191.4367, Y 36.6188, Z -4.6667, A 0.000, B 0.000, C 0.000 }
gfCNCPoint4[382] = {X 192.6036, Y 35.8984, Z -4.6667, A 0.000, B 0.000, C 0.000 }
gfCNCPoint4[383] = {X 192.6773, Y 35.2163, Z -4.6667, A 0.000, B 0.000, C 0.000 }
gfCNCPoint4[384] = {X 192.8600, Y 34.5550, Z -4.6667, A 0.000, B 0.000, C 0.000 }
gfCNCPoint4[385] = {X 193.1469, Y 33.9318, Z -4.6667, A 0.000, B 0.000, C 0.000 }
gfCNCPoint4[386] = {X 192.7149, Y 34.0342, Z -4.6667, A 0.000, B 0.000, C 0.000 }
gfCNCPoint4[387] = {X 190.9731, Y 34.3101, Z -4.6667, A 0.000, B 0.000, C 0.000 }
gfCNCPoint4[388] = {X 189.2183, Y 34.4844, Z -4.6667, A 0.000, B 0.000, C 0.000 }
gfCNCPoint4[389] = {X 186.9528, Y 34.6235, Z -4.6667, A 0.000, B 0.000, C 0.000 }
gfCNCPoint4[390] = {X 182.9969, Y 35.2157, Z -4.6667, A 0.000, B 0.000, C 0.000 }
gfCNCPoint4[391] = {X 190.9466, Y 34.6475, Z -4.6667, A 0.000, B 0.000, C 0.000 }
gfCNCPoint4[392] = {X 186.9479, Y 34.5437, Z -4.6667, A 0.000, B 0.000, C 0.000 }
gfCNCPoint4[393] = {X 182.5608, Y 34.8131, Z -4.6667, A 0.000, B 0.000, C 0.000 }
gfCNCPoint4[394] = {X 181.7089, Y 34.9154, Z -4.6667, A 0.000, B 0.000, C 0.000 }
gfCNCPoint4[395] = {X 180.8747, Y 35.1158, Z -4.6667, A 0.000, B 0.000, C 0.000 }
gfCNCPoint4[396] = {X 180.8337, Y 35.2842, Z -4.6667, A 0.000, B 0.000, C 0.000 }
gfCNCPoint4[397] = {X 180.8247, Y 35.4572, Z -4.6667, A 0.000, B 0.000, C 0.000 }
gfCNCPoint4[398] = {X 180.9301, Y 36.0765, Z -4.6667, A 0.000, B 0.000, C 0.000 }
gfCNCPoint4[399] = {X 181.2234, Y 36.6320, Z -4.6667, A 0.000, B 0.000, C 0.000 }
gfCNCPoint4[400] = {X 181.6754, Y 37.0683, Z -4.6667, A 0.000, B 0.000, C 0.000 }
gfCNCPoint4[401] = {X 182.3240, Y 37.4390, Z -4.6667, A 0.000, B 0.000, C 0.000 }
gfCNCPoint4[402] = {X 183.0176, Y 37.7168, Z -4.6667, A 0.000, B 0.000, C 0.000 }
gfCNCPoint4[403] = {X 184.4567, Y 38.0383, Z -4.6667, A 0.000, B 0.000, C 0.000 }
gfCNCPoint4[404] = {X 185.9265, Y 38.1572, Z -4.6667, A 0.000, B 0.000, C 0.000 }
gfCNCPoint4[405] = {X 187.3986, Y 38.0712, Z -4.6667, A 0.000, B 0.000, C 0.000 }
gfCNCPoint4[406] = {X 188.8445, Y 37.7820, Z -4.6667, A 0.000, B 0.000, C 0.000 }
gfCNCPoint4[407] = {X 190.2364, Y 37.2951, Z -4.6667, A 0.000, B 0.000, C 0.000 }
gfCNCPoint4[408] = {X 191.4933, Y 36.6789, Z -4.6667, A 0.000, B 0.000, C 0.000 }
gfCNCPoint4[409] = {X 192.6827, Y 35.9410, Z -4.6667, A 0.000, B 0.000, C 0.000 }
gfCNCPoint4[410] = {X 192.7626, Y 35.1968, Z -4.6667, A 0.000, B 0.000, C 0.000 }
gfCNCPoint4[411] = {X 192.9746, Y 34.4788, Z -4.6667, A 0.000, B 0.000, C 0.000 }
gfCNCPoint4[412] = {X 193.3118, Y 33.8105, Z -4.6667, A 0.000, B 0.000, C 0.000 }
gfCNCPoint4[413] = {X 192.6983, Y 33.9560, Z -4.6667, A 0.000, B 0.000, C 0.000 }
gfCNCPoint4[414] = {X 190.9622, Y 34.2309, Z -4.6667, A 0.000, B 0.000, C 0.000 }
gfCNCPoint4[415] = {X 189.2131, Y 34.4046, Z -4.6667, A 0.000, B 0.000, C 0.000 }
gfCNCPoint4[416] = {X 186.9479, Y 34.5437, Z -4.6667, A 0.000, B 0.000, C 0.000 }
gfCNCPoint4[417] = {X 182.9920, Y 35.1359, Z -4.6667, A 0.000, B 0.000, C 0.000 }
gfCNCPoint4[418] = {X 190.9417, Y 34.5676, Z -4.6667, A 0.000, B 0.000, C 0.000 }
gfCNCPoint4[419] = {X 186.9430, Y 34.4638, Z -4.6667, A 0.000, B 0.000, C 0.000 }
gfCNCPoint4[420] = {X 182.5559, Y 34.7332, Z -4.6667, A 0.000, B 0.000, C 0.000 }
gfCNCPoint4[421] = {X 181.6752, Y 34.8402, Z -4.6667, A 0.000, B 0.000, C 0.000 }
gfCNCPoint4[422] = {X 180.8134, Y 35.0509, Z -4.6667, A 0.000, B 0.000, C 0.000 }
gfCNCPoint4[423] = {X 180.7578, Y 35.2515, Z -4.6667, A 0.000, B 0.000, C 0.000 }
gfCNCPoint4[424] = {X 180.7448, Y 35.4593, Z -4.6667, A 0.000, B 0.000, C 0.000 }
gfCNCPoint4[425] = {X 180.8547, Y 36.1033, Z -4.6667, A 0.000, B 0.000, C 0.000 }
gfCNCPoint4[426] = {X 181.1601, Y 36.6809, Z -4.6667, A 0.000, B 0.000, C 0.000 }
gfCNCPoint4[427] = {X 181.6303, Y 37.1344, Z -4.6667, A 0.000, B 0.000, C 0.000 }
gfCNCPoint4[428] = {X 182.2893, Y 37.5111, Z -4.6667, A 0.000, B 0.000, C 0.000 }
gfCNCPoint4[429] = {X 182.9939, Y 37.7932, Z -4.6667, A 0.000, B 0.000, C 0.000 }
gfCNCPoint4[430] = {X 184.4440, Y 38.1173, Z -4.6667, A 0.000, B 0.000, C 0.000 }
gfCNCPoint4[431] = {X 185.9251, Y 38.2372, Z -4.6667, A 0.000, B 0.000, C 0.000 }
gfCNCPoint4[432] = {X 187.4084, Y 38.1506, Z -4.6667, A 0.000, B 0.000, C 0.000 }
gfCNCPoint4[433] = {X 188.8655, Y 37.8592, Z -4.6667, A 0.000, B 0.000, C 0.000 }
gfCNCPoint4[434] = {X 190.2680, Y 37.3685, Z -4.6667, A 0.000, B 0.000, C 0.000 }
gfCNCPoint4[435] = {X 191.5501, Y 36.7389, Z -4.6667, A 0.000, B 0.000, C 0.000 }
gfCNCPoint4[436] = {X 192.7622, Y 35.9833, Z -4.6667, A 0.000, B 0.000, C 0.000 }
gfCNCPoint4[437] = {X 192.8358, Y 35.2391, Z -4.6667, A 0.000, B 0.000, C 0.000 }
gfCNCPoint4[438] = {X 193.0440, Y 34.5210, Z -4.6667, A 0.000, B 0.000, C 0.000 }
gfCNCPoint4[439] = {X 193.3797, Y 33.8528, Z -4.6667, A 0.000, B 0.000, C 0.000 }
gfCNCPoint4[440] = {X 193.4227, Y 33.7853, Z -4.6667, A 0.000, B 0.000, C 0.000 }
gfCNCPoint4[441] = {X 193.4670, Y 33.7186, Z -4.6667, A 0.000, B 0.000, C 0.000 }
gfCNCPoint4[442] = {X 193.3656, Y 33.7155, Z -4.6667, A 0.000, B 0.000, C 0.000 }
gfCNCPoint4[443] = {X 192.6816, Y 33.8777, Z -4.6667, A 0.000, B 0.000, C 0.000 }
gfCNCPoint4[444] = {X 190.9512, Y 34.1516, Z -4.6667, A 0.000, B 0.000, C 0.000 }
gfCNCPoint4[445] = {X 189.2078, Y 34.3248, Z -4.6667, A 0.000, B 0.000, C 0.000 }
gfCNCPoint4[446] = {X 186.9430, Y 34.4638, Z -4.6667, A 0.000, B 0.000, C 0.000 }
gfCNCPoint4[447] = {X 182.9871, Y 35.0560, Z -4.6667, A 0.000, B 0.000, C 0.000 }
gfCNCPoint4[448] = {X 190.9306, Y 34.1389, Z -4.6667, A 0.000, B 0.000, C 0.000 }
gfCNCPoint4[449] = {X 186.9381, Y 34.3840, Z -4.6667, A 0.000, B 0.000, C 0.000 }
gfCNCPoint4[450] = {X 182.5510, Y 34.6534, Z -4.6667, A 0.000, B 0.000, C 0.000 }
gfCNCPoint4[451] = {X 181.6423, Y 34.7649, Z -4.6667, A 0.000, B 0.000, C 0.000 }
gfCNCPoint4[452] = {X 180.7539, Y 34.9857, Z -4.6667, A 0.000, B 0.000, C 0.000 }
gfCNCPoint4[453] = {X 180.6824, Y 35.2185, Z -4.6667, A 0.000, B 0.000, C 0.000 }
gfCNCPoint4[454] = {X 180.6648, Y 35.4613, Z -4.6667, A 0.000, B 0.000, C 0.000 }
gfCNCPoint4[455] = {X 180.7793, Y 36.1300, Z -4.6667, A 0.000, B 0.000, C 0.000 }
gfCNCPoint4[456] = {X 181.0967, Y 36.7297, Z -4.6667, A 0.000, B 0.000, C 0.000 }
gfCNCPoint4[457] = {X 181.5852, Y 37.2005, Z -4.6667, A 0.000, B 0.000, C 0.000 }
gfCNCPoint4[458] = {X 182.2545, Y 37.5831, Z -4.6667, A 0.000, B 0.000, C 0.000 }
gfCNCPoint4[459] = {X 182.9702, Y 37.8696, Z -4.6667, A 0.000, B 0.000, C 0.000 }
gfCNCPoint4[460] = {X 184.4313, Y 38.1963, Z -4.6667, A 0.000, B 0.000, C 0.000 }
gfCNCPoint4[461] = {X 185.9236, Y 38.3172, Z -4.6667, A 0.000, B 0.000, C 0.000 }
gfCNCPoint4[462] = {X 187.4183, Y 38.2300, Z -4.6667, A 0.000, B 0.000, C 0.000 }
gfCNCPoint4[463] = {X 188.8864, Y 37.9364, Z -4.6667, A 0.000, B 0.000, C 0.000 }
gfCNCPoint4[464] = {X 190.2996, Y 37.4420, Z -4.6667, A 0.000, B 0.000, C 0.000 }
gfCNCPoint4[465] = {X 191.6072, Y 36.7987, Z -4.6667, A 0.000, B 0.000, C 0.000 }
gfCNCPoint4[466] = {X 192.8422, Y 36.0250, Z -4.6667, A 0.000, B 0.000, C 0.000 }
gfCNCPoint4[467] = {X 192.9290, Y 35.1818, Z -4.6667, A 0.000, B 0.000, C 0.000 }
gfCNCPoint4[468] = {X 193.1917, Y 34.3757, Z -4.6667, A 0.000, B 0.000, C 0.000 }
gfCNCPoint4[469] = {X 193.6183, Y 33.6431, Z -4.6667, A 0.000, B 0.000, C 0.000 }
gfCNCPoint4[470] = {X 193.3575, Y 33.6352, Z -4.6667, A 0.000, B 0.000, C 0.000 }
gfCNCPoint4[471] = {X 192.6650, Y 33.7994, Z -4.6667, A 0.000, B 0.000, C 0.000 }
gfCNCPoint4[472] = {X 190.9402, Y 34.0724, Z -4.6667, A 0.000, B 0.000, C 0.000 }
gfCNCPoint4[473] = {X 189.2026, Y 34.2450, Z -4.6667, A 0.000, B 0.000, C 0.000 }
gfCNCPoint4[474] = {X 186.9381, Y 34.3840, Z -4.6667, A 0.000, B 0.000, C 0.000 }
gfCNCPoint4[475] = {X 182.9456, Y 34.6291, Z -4.6667, A 0.000, B 0.000, C 0.000 }
gfCNCPoint4[476] = {X 182.9456, Y 34.6291, Z -1.6667, A 0.000, B 0.000, C 0.000 }
gfCNCPoint4[477] = {X 182.9456, Y 34.6291, Z 11.0000, A 0.000, B 0.000, C 0.000 }
gfCNCPoint4[478] = {X 165.6772, Y 73.8165, Z 11.0000, A 0.000, B 0.000, C 0.000 }
gfCNCPoint4[479] = {X 165.6772, Y 73.8165, Z -0.8333, A 0.000, B 0.000, C 0.000 }
gfCNCPoint4[480] = {X 161.3996, Y 78.5670, Z -2.5462, A 0.000, B 0.000, C 0.000 }
gfCNCPoint4[481] = {X 169.3132, Y 78.5670, Z -4.6667, A 0.000, B 0.000, C 0.000 }
gfCNCPoint4[482] = {X 169.3132, Y 76.1670, Z -4.6667, A 0.000, B 0.000, C 0.000 }
gfCNCPoint4[483] = {X 171.8361, Y 76.1670, Z -4.6667, A 0.000, B 0.000, C 0.000 }
gfCNCPoint4[484] = {X 169.3147, Y 73.3634, Z -4.6667, A 0.000, B 0.000, C 0.000 }
gfCNCPoint4[485] = {X 166.7903, Y 76.1670, Z -4.6667, A 0.000, B 0.000, C 0.000 }
gfCNCPoint4[486] = {X 169.3132, Y 76.1670, Z -4.6667, A 0.000, B 0.000, C 0.000 }
gfCNCPoint4[487] = {X 169.3132, Y 78.5670, Z -4.6667, A 0.000, B 0.000, C 0.000 }
gfCNCPoint4[488] = {X 177.2224, Y 78.5670, Z -4.6667, A 0.000, B 0.000, C 0.000 }
gfCNCPoint4[489] = {X 169.3158, Y 69.7756, Z -4.6667, A 0.000, B 0.000, C 0.000 }
gfCNCPoint4[490] = {X 161.3996, Y 78.5670, Z -4.6667, A 0.000, B 0.000, C 0.000 }
gfCNCPoint4[491] = {X 169.3132, Y 78.5670, Z -4.6667, A 0.000, B 0.000, C 0.000 }
gfCNCPoint4[492] = {X 169.3132, Y 74.6470, Z -4.6667, A 0.000, B 0.000, C 0.000 }
gfCNCPoint4[493] = {X 169.3132, Y 78.6470, Z -4.6667, A 0.000, B 0.000, C 0.000 }
gfCNCPoint4[494] = {X 177.4019, Y 78.6470, Z -4.6667, A 0.000, B 0.000, C 0.000 }
gfCNCPoint4[495] = {X 169.3159, Y 69.6560, Z -4.6667, A 0.000, B 0.000, C 0.000 }
gfCNCPoint4[496] = {X 161.2199, Y 78.6470, Z -4.6667, A 0.000, B 0.000, C 0.000 }
gfCNCPoint4[497] = {X 169.3132, Y 78.6470, Z -4.6667, A 0.000, B 0.000, C 0.000 }
gfCNCPoint4[498] = {X 169.3132, Y 74.6470, Z -4.6667, A 0.000, B 0.000, C 0.000 }
gfCNCPoint4[499] = {X 169.3132, Y 74.7270, Z -4.6667, A 0.000, B 0.000, C 0.000 }
gfCNCPoint4[500] = {X 169.3132, Y 78.7270, Z -4.6667, A 0.000, B 0.000, C 0.000 }
gfCNCPoint4[501] = {X 177.5814, Y 78.7270, Z -4.6667, A 0.000, B 0.000, C 0.000 }
gfCNCPoint4[502] = {X 169.3159, Y 69.5364, Z -4.6667, A 0.000, B 0.000, C 0.000 }
gfCNCPoint4[503] = {X 161.0403, Y 78.7270, Z -4.6667, A 0.000, B 0.000, C 0.000 }
gfCNCPoint4[504] = {X 169.3132, Y 78.7270, Z -4.6667, A 0.000, B 0.000, C 0.000 }
gfCNCPoint4[505] = {X 169.3132, Y 74.7270, Z -4.6667, A 0.000, B 0.000, C 0.000 }
gfCNCPoint4[506] = {X 169.3132, Y 74.8070, Z -4.6667, A 0.000, B 0.000, C 0.000 }
gfCNCPoint4[507] = {X 169.3132, Y 78.8070, Z -4.6667, A 0.000, B 0.000, C 0.000 }
gfCNCPoint4[508] = {X 177.7610, Y 78.8070, Z -4.6667, A 0.000, B 0.000, C 0.000 }
gfCNCPoint4[509] = {X 169.3159, Y 69.4168, Z -4.6667, A 0.000, B 0.000, C 0.000 }
gfCNCPoint4[510] = {X 160.8606, Y 78.8070, Z -4.6667, A 0.000, B 0.000, C 0.000 }
gfCNCPoint4[511] = {X 169.3132, Y 78.8070, Z -4.6667, A 0.000, B 0.000, C 0.000 }
gfCNCPoint4[512] = {X 169.3132, Y 74.8070, Z -4.6667, A 0.000, B 0.000, C 0.000 }
gfCNCPoint4[513] = {X 169.3132, Y 74.8870, Z -4.6667, A 0.000, B 0.000, C 0.000 }
gfCNCPoint4[514] = {X 169.3132, Y 78.8870, Z -4.6667, A 0.000, B 0.000, C 0.000 }
gfCNCPoint4[515] = {X 177.9405, Y 78.8870, Z -4.6667, A 0.000, B 0.000, C 0.000 }
gfCNCPoint4[516] = {X 169.3160, Y 69.2972, Z -4.6667, A 0.000, B 0.000, C 0.000 }
gfCNCPoint4[517] = {X 160.6809, Y 78.8870, Z -4.6667, A 0.000, B 0.000, C 0.000 }
gfCNCPoint4[518] = {X 169.3132, Y 78.8870, Z -4.6667, A 0.000, B 0.000, C 0.000 }
gfCNCPoint4[519] = {X 169.3132, Y 74.8870, Z -4.6667, A 0.000, B 0.000, C 0.000 }
gfCNCPoint4[520] = {X 169.3132, Y 74.9670, Z -4.6667, A 0.000, B 0.000, C 0.000 }
gfCNCPoint4[521] = {X 169.3132, Y 78.9670, Z -4.6667, A 0.000, B 0.000, C 0.000 }
gfCNCPoint4[522] = {X 178.1201, Y 78.9670, Z -4.6667, A 0.000, B 0.000, C 0.000 }
gfCNCPoint4[523] = {X 169.3160, Y 69.1776, Z -4.6667, A 0.000, B 0.000, C 0.000 }
gfCNCPoint4[524] = {X 160.5012, Y 78.9670, Z -4.6667, A 0.000, B 0.000, C 0.000 }
gfCNCPoint4[525] = {X 169.3132, Y 78.9670, Z -4.6667, A 0.000, B 0.000, C 0.000 }
gfCNCPoint4[526] = {X 169.3132, Y 74.9670, Z -4.6667, A 0.000, B 0.000, C 0.000 }
gfCNCPoint4[527] = {X 169.3132, Y 74.9670, Z -1.6667, A 0.000, B 0.000, C 0.000 }
gfCNCPoint4[528] = {X 169.3132, Y 74.9670, Z 11.0000, A 0.000, B 0.000, C 0.000 }
gfCNCPoint4[529] = {X 11.7100, Y 37.8789, Z 11.0000, A 0.000, B 0.000, C 0.000 }
gfCNCPoint4[530] = {X 11.7100, Y 37.8789, Z -0.8333, A 0.000, B 0.000, C 0.000 }
gfCNCPoint4[531] = {X 12.4890, Y 37.9507, Z -1.0430, A 0.000, B 0.000, C 0.000 }
gfCNCPoint4[532] = {X 14.1304, Y 37.8411, Z -1.4838, A 0.000, B 0.000, C 0.000 }
gfCNCPoint4[533] = {X 15.7339, Y 37.4736, Z -1.9245, A 0.000, B 0.000, C 0.000 }
gfCNCPoint4[534] = {X 16.4661, Y 37.1806, Z -2.1359, A 0.000, B 0.000, C 0.000 }
gfCNCPoint4[535] = {X 17.2988, Y 36.8474, Z -2.3762, A 0.000, B 0.000, C 0.000 }
gfCNCPoint4[536] = {X 18.2934, Y 36.3175, Z -2.6781, A 0.000, B 0.000, C 0.000 }
gfCNCPoint4[537] = {X 19.0345, Y 35.8123, Z -2.9185, A 0.000, B 0.000, C 0.000 }
gfCNCPoint4[538] = {X 19.0577, Y 35.2981, Z -3.0564, A 0.000, B 0.000, C 0.000 }
gfCNCPoint4[539] = {X 19.2190, Y 34.6354, Z -3.2391, A 0.000, B 0.000, C 0.000 }
gfCNCPoint4[540] = {X 19.4345, Y 34.1680, Z -3.3770, A 0.000, B 0.000, C 0.000 }
gfCNCPoint4[541] = {X 18.1999, Y 34.4164, Z -3.7145, A 0.000, B 0.000, C 0.000 }
gfCNCPoint4[542] = {X 17.3668, Y 34.5296, Z -3.9398, A 0.000, B 0.000, C 0.000 }
gfCNCPoint4[543] = {X 16.1107, Y 34.6196, Z -4.2772, A 0.000, B 0.000, C 0.000 }
gfCNCPoint4[544] = {X 15.3859, Y 34.6733, Z -4.4719, A 0.000, B 0.000, C 0.000 }
gfCNCPoint4[545] = {X 14.6609, Y 34.7229, Z -4.6667, A 0.000, B 0.000, C 0.000 }
gfCNCPoint4[546] = {X 12.2607, Y 34.8755, Z -4.6667, A 0.000, B 0.000, C 0.000 }
gfCNCPoint4[547] = {X 9.8592, Y 35.0052, Z -4.6667, A 0.000, B 0.000, C 0.000 }
gfCNCPoint4[548] = {X 8.7536, Y 35.0953, Z -4.6667, A 0.000, B 0.000, C 0.000 }
gfCNCPoint4[549] = {X 7.6651, Y 35.3093, Z -4.6667, A 0.000, B 0.000, C 0.000 }
gfCNCPoint4[550] = {X 7.6556, Y 35.3710, Z -4.6667, A 0.000, B 0.000, C 0.000 }
gfCNCPoint4[551] = {X 7.6522, Y 35.4334, Z -4.6667, A 0.000, B 0.000, C 0.000 }
gfCNCPoint4[552] = {X 7.7530, Y 36.0263, Z -4.6667, A 0.000, B 0.000, C 0.000 }
gfCNCPoint4[553] = {X 8.0476, Y 36.5506, Z -4.6667, A 0.000, B 0.000, C 0.000 }
gfCNCPoint4[554] = {X 8.5016, Y 36.9451, Z -4.6667, A 0.000, B 0.000, C 0.000 }
gfCNCPoint4[555] = {X 9.2694, Y 37.3346, Z -4.6667, A 0.000, B 0.000, C 0.000 }
gfCNCPoint4[556] = {X 10.0863, Y 37.6066, Z -4.6667, A 0.000, B 0.000, C 0.000 }
gfCNCPoint4[557] = {X 11.3634, Y 37.8449, Z -4.6667, A 0.000, B 0.000, C 0.000 }
gfCNCPoint4[558] = {X 12.6604, Y 37.9215, Z -4.6667, A 0.000, B 0.000, C 0.000 }
gfCNCPoint4[559] = {X 13.9567, Y 37.8349, Z -4.6667, A 0.000, B 0.000, C 0.000 }
gfCNCPoint4[560] = {X 15.2320, Y 37.5867, Z -4.6667, A 0.000, B 0.000, C 0.000 }
gfCNCPoint4[561] = {X 16.4661, Y 37.1806, Z -4.6667, A 0.000, B 0.000, C 0.000 }
gfCNCPoint4[562] = {X 17.7876, Y 36.5664, Z -4.6667, A 0.000, B 0.000, C 0.000 }
gfCNCPoint4[563] = {X 19.0345, Y 35.8123, Z -4.6667, A 0.000, B 0.000, C 0.000 }
gfCNCPoint4[564] = {X 19.1547, Y 34.9707, Z -4.6667, A 0.000, B 0.000, C 0.000 }
gfCNCPoint4[565] = {X 19.4345, Y 34.1680, Z -4.6667, A 0.000, B 0.000, C 0.000 }
gfCNCPoint4[566] = {X 17.7798, Y 34.4466, Z -4.6667, A 0.000, B 0.000, C 0.000 }
gfCNCPoint4[567] = {X 16.1107, Y 34.6196, Z -4.6667, A 0.000, B 0.000, C 0.000 }
gfCNCPoint4[568] = {X 15.3859, Y 34.6723, Z -4.6667, A 0.000, B 0.000, C 0.000 }
gfCNCPoint4[569] = {X 14.6609, Y 34.7229, Z -4.6667, A 0.000, B 0.000, C 0.000 }
gfCNCPoint4[570] = {X 18.6547, Y 34.7190, Z -4.6667, A 0.000, B 0.000, C 0.000 }
gfCNCPoint4[571] = {X 14.6555, Y 34.6431, Z -4.6667, A 0.000, B 0.000, C 0.000 }
gfCNCPoint4[572] = {X 12.2589, Y 34.7955, Z -4.6667, A 0.000, B 0.000, C 0.000 }
gfCNCPoint4[573] = {X 9.8611, Y 34.9251, Z -4.6667, A 0.000, B 0.000, C 0.000 }
gfCNCPoint4[574] = {X 8.7208, Y 35.0191, Z -4.6667, A 0.000, B 0.000, C 0.000 }
gfCNCPoint4[575] = {X 7.5989, Y 35.2438, Z -4.6667, A 0.000, B 0.000, C 0.000 }
gfCNCPoint4[576] = {X 7.5791, Y 35.3375, Z -4.6667, A 0.000, B 0.000, C 0.000 }
gfCNCPoint4[577] = {X 7.5722, Y 35.4331, Z -4.6667, A 0.000, B 0.000, C 0.000 }
gfCNCPoint4[578] = {X 7.6776, Y 36.0530, Z -4.6667, A 0.000, B 0.000, C 0.000 }
gfCNCPoint4[579] = {X 7.9856, Y 36.6011, Z -4.6667, A 0.000, B 0.000, C 0.000 }
gfCNCPoint4[580] = {X 8.4602, Y 37.0135, Z -4.6667, A 0.000, B 0.000, C 0.000 }
gfCNCPoint4[581] = {X 9.2386, Y 37.4084, Z -4.6667, A 0.000, B 0.000, C 0.000 }
gfCNCPoint4[582] = {X 10.0667, Y 37.6841, Z -4.6667, A 0.000, B 0.000, C 0.000 }
gfCNCPoint4[583] = {X 11.3537, Y 37.9243, Z -4.6667, A 0.000, B 0.000, C 0.000 }
gfCNCPoint4[584] = {X 12.6607, Y 38.0015, Z -4.6667, A 0.000, B 0.000, C 0.000 }
gfCNCPoint4[585] = {X 13.9670, Y 37.9143, Z -4.6667, A 0.000, B 0.000, C 0.000 }
gfCNCPoint4[586] = {X 15.2522, Y 37.6641, Z -4.6667, A 0.000, B 0.000, C 0.000 }
gfCNCPoint4[587] = {X 16.4959, Y 37.2549, Z -4.6667, A 0.000, B 0.000, C 0.000 }
gfCNCPoint4[588] = {X 17.8430, Y 36.6275, Z -4.6667, A 0.000, B 0.000, C 0.000 }
gfCNCPoint4[589] = {X 19.1128, Y 35.8556, Z -4.6667, A 0.000, B 0.000, C 0.000 }
gfCNCPoint4[590] = {X 19.2471, Y 34.9312, Z -4.6667, A 0.000, B 0.000, C 0.000 }
gfCNCPoint4[591] = {X 19.5770, Y 34.0573, Z -4.6667, A 0.000, B 0.000, C 0.000 }
gfCNCPoint4[592] = {X 17.8490, Y 34.3563, Z -4.6667, A 0.000, B 0.000, C 0.000 }
gfCNCPoint4[593] = {X 16.1048, Y 34.5398, Z -4.6667, A 0.000, B 0.000, C 0.000 }
gfCNCPoint4[594] = {X 15.3802, Y 34.5925, Z -4.6667, A 0.000, B 0.000, C 0.000 }
gfCNCPoint4[595] = {X 14.6555, Y 34.6431, Z -4.6667, A 0.000, B 0.000, C 0.000 }
gfCNCPoint4[596] = {X 10.7038, Y 35.2627, Z -4.6667, A 0.000, B 0.000, C 0.000 }
gfCNCPoint4[597] = {X 18.6493, Y 34.6392, Z -4.6667, A 0.000, B 0.000, C 0.000 }
gfCNCPoint4[598] = {X 14.6500, Y 34.5633, Z -4.6667, A 0.000, B 0.000, C 0.000 }
gfCNCPoint4[599] = {X 12.2547, Y 34.7156, Z -4.6667, A 0.000, B 0.000, C 0.000 }
gfCNCPoint4[600] = {X 9.8581, Y 34.8452, Z -4.6667, A 0.000, B 0.000, C 0.000 }
gfCNCPoint4[601] = {X 8.6872, Y 34.9431, Z -4.6667, A 0.000, B 0.000, C 0.000 }
gfCNCPoint4[602] = {X 7.5359, Y 35.1777, Z -4.6667, A 0.000, B 0.000, C 0.000 }
gfCNCPoint4[603] = {X 7.5035, Y 35.3034, Z -4.6667, A 0.000, B 0.000, C 0.000 }
gfCNCPoint4[604] = {X 7.4922, Y 35.4328, Z -4.6667, A 0.000, B 0.000, C 0.000 }
gfCNCPoint4[605] = {X 7.6022, Y 36.0797, Z -4.6667, A 0.000, B 0.000, C 0.000 }
gfCNCPoint4[606] = {X 7.9236, Y 36.6517, Z -4.6667, A 0.000, B 0.000, C 0.000 }
gfCNCPoint4[607] = {X 8.4189, Y 37.0820, Z -4.6667, A 0.000, B 0.000, C 0.000 }
gfCNCPoint4[608] = {X 9.2078, Y 37.4822, Z -4.6667, A 0.000, B 0.000, C 0.000 }
gfCNCPoint4[609] = {X 10.0471, Y 37.7617, Z -4.6667, A 0.000, B 0.000, C 0.000 }
gfCNCPoint4[610] = {X 11.3440, Y 38.0038, Z -4.6667, A 0.000, B 0.000, C 0.000 }
gfCNCPoint4[611] = {X 12.6610, Y 38.0815, Z -4.6667, A 0.000, B 0.000, C 0.000 }
gfCNCPoint4[612] = {X 13.9774, Y 37.9936, Z -4.6667, A 0.000, B 0.000, C 0.000 }
gfCNCPoint4[613] = {X 15.2724, Y 37.7415, Z -4.6667, A 0.000, B 0.000, C 0.000 }
gfCNCPoint4[614] = {X 16.5256, Y 37.3292, Z -4.6667, A 0.000, B 0.000, C 0.000 }
gfCNCPoint4[615] = {X 17.8986, Y 36.6885, Z -4.6667, A 0.000, B 0.000, C 0.000 }
gfCNCPoint4[616] = {X 19.1915, Y 35.8986, Z -4.6667, A 0.000, B 0.000, C 0.000 }
gfCNCPoint4[617] = {X 19.2643, Y 35.2208, Z -4.6667, A 0.000, B 0.000, C 0.000 }
gfCNCPoint4[618] = {X 19.4447, Y 34.5635, Z -4.6667, A 0.000, B 0.000, C 0.000 }
gfCNCPoint4[619] = {X 19.7282, Y 33.9436, Z -4.6667, A 0.000, B 0.000, C 0.000 }
gfCNCPoint4[620] = {X 17.9226, Y 34.2652, Z -4.6667, A 0.000, B 0.000, C 0.000 }
gfCNCPoint4[621] = {X 16.0990, Y 34.4600, Z -4.6667, A 0.000, B 0.000, C 0.000 }
gfCNCPoint4[622] = {X 15.3746, Y 34.5127, Z -4.6667, A 0.000, B 0.000, C 0.000 }
gfCNCPoint4[623] = {X 14.6500, Y 34.5633, Z -4.6667, A 0.000, B 0.000, C 0.000 }
gfCNCPoint4[624] = {X 10.6983, Y 35.1829, Z -4.6667, A 0.000, B 0.000, C 0.000 }
gfCNCPoint4[625] = {X 18.6438, Y 34.5594, Z -4.6667, A 0.000, B 0.000, C 0.000 }
gfCNCPoint4[626] = {X 14.6445, Y 34.4835, Z -4.6667, A 0.000, B 0.000, C 0.000 }
gfCNCPoint4[627] = {X 12.2505, Y 34.6357, Z -4.6667, A 0.000, B 0.000, C 0.000 }
gfCNCPoint4[628] = {X 9.8551, Y 34.7652, Z -4.6667, A 0.000, B 0.000, C 0.000 }
gfCNCPoint4[629] = {X 8.6550, Y 34.8669, Z -4.6667, A 0.000, B 0.000, C 0.000 }
gfCNCPoint4[630] = {X 7.4756, Y 35.1110, Z -4.6667, A 0.000, B 0.000, C 0.000 }
gfCNCPoint4[631] = {X 7.4285, Y 35.2687, Z -4.6667, A 0.000, B 0.000, C 0.000 }
gfCNCPoint4[632] = {X 7.4122, Y 35.4325, Z -4.6667, A 0.000, B 0.000, C 0.000 }
gfCNCPoint4[633] = {X 7.5267, Y 36.1064, Z -4.6667, A 0.000, B 0.000, C 0.000 }
gfCNCPoint4[634] = {X 7.8615, Y 36.7022, Z -4.6667, A 0.000, B 0.000, C 0.000 }
gfCNCPoint4[635] = {X 8.3775, Y 37.1505, Z -4.6667, A 0.000, B 0.000, C 0.000 }
gfCNCPoint4[636] = {X 9.1770, Y 37.5561, Z -4.6667, A 0.000, B 0.000, C 0.000 }
gfCNCPoint4[637] = {X 10.0275, Y 37.8393, Z -4.6667, A 0.000, B 0.000, C 0.000 }
gfCNCPoint4[638] = {X 11.3343, Y 38.0832, Z -4.6667, A 0.000, B 0.000, C 0.000 }
gfCNCPoint4[639] = {X 12.6613, Y 38.1615, Z -4.6667, A 0.000, B 0.000, C 0.000 }
gfCNCPoint4[640] = {X 13.9877, Y 38.0729, Z -4.6667, A 0.000, B 0.000, C 0.000 }
gfCNCPoint4[641] = {X 15.2926, Y 37.8189, Z -4.6667, A 0.000, B 0.000, C 0.000 }
gfCNCPoint4[642] = {X 16.5553, Y 37.4034, Z -4.6667, A 0.000, B 0.000, C 0.000 }
gfCNCPoint4[643] = {X 17.9544, Y 36.7493, Z -4.6667, A 0.000, B 0.000, C 0.000 }
gfCNCPoint4[644] = {X 19.2706, Y 35.9411, Z -4.6667, A 0.000, B 0.000, C 0.000 }
gfCNCPoint4[645] = {X 19.3492, Y 35.2030, Z -4.6667, A 0.000, B 0.000, C 0.000 }
gfCNCPoint4[646] = {X 19.5578, Y 34.4905, Z -4.6667, A 0.000, B 0.000, C 0.000 }
gfCNCPoint4[647] = {X 19.8897, Y 33.8265, Z -4.6667, A 0.000, B 0.000, C 0.000 }
gfCNCPoint4[648] = {X 18.0016, Y 34.1730, Z -4.6667, A 0.000, B 0.000, C 0.000 }
gfCNCPoint4[649] = {X 16.0932, Y 34.3802, Z -4.6667, A 0.000, B 0.000, C 0.000 }
gfCNCPoint4[650] = {X 15.3690, Y 34.4329, Z -4.6667, A 0.000, B 0.000, C 0.000 }
gfCNCPoint4[651] = {X 14.6445, Y 34.4835, Z -4.6667, A 0.000, B 0.000, C 0.000 }
gfCNCPoint4[652] = {X 10.6928, Y 35.1031, Z -4.6667, A 0.000, B 0.000, C 0.000 }
gfCNCPoint4[653] = {X 18.6384, Y 34.4796, Z -4.6667, A 0.000, B 0.000, C 0.000 }
gfCNCPoint4[654] = {X 14.6391, Y 34.4036, Z -4.6667, A 0.000, B 0.000, C 0.000 }
gfCNCPoint4[655] = {X 12.2463, Y 34.5558, Z -4.6667, A 0.000, B 0.000, C 0.000 }
gfCNCPoint4[656] = {X 9.8522, Y 34.6853, Z -4.6667, A 0.000, B 0.000, C 0.000 }
gfCNCPoint4[657] = {X 8.6239, Y 34.7906, Z -4.6667, A 0.000, B 0.000, C 0.000 }
gfCNCPoint4[658] = {X 7.4174, Y 35.0439, Z -4.6667, A 0.000, B 0.000, C 0.000 }
gfCNCPoint4[659] = {X 7.3541, Y 35.2336, Z -4.6667, A 0.000, B 0.000, C 0.000 }
gfCNCPoint4[660] = {X 7.3322, Y 35.4323, Z -4.6667, A 0.000, B 0.000, C 0.000 }
gfCNCPoint4[661] = {X 7.3990, Y 35.9623, Z -4.6667, A 0.000, B 0.000, C 0.000 }
gfCNCPoint4[662] = {X 7.5987, Y 36.4579, Z -4.6667, A 0.000, B 0.000, C 0.000 }
gfCNCPoint4[663] = {X 7.9181, Y 36.8862, Z -4.6667, A 0.000, B 0.000, C 0.000 }
gfCNCPoint4[664] = {X 8.3361, Y 37.2189, Z -4.6667, A 0.000, B 0.000, C 0.000 }
gfCNCPoint4[665] = {X 9.1461, Y 37.6299, Z -4.6667, A 0.000, B 0.000, C 0.000 }
gfCNCPoint4[666] = {X 10.0079, Y 37.9168, Z -4.6667, A 0.000, B 0.000, C 0.000 }
gfCNCPoint4[667] = {X 11.3246, Y 38.1626, Z -4.6667, A 0.000, B 0.000, C 0.000 }
gfCNCPoint4[668] = {X 12.6616, Y 38.2415, Z -4.6667, A 0.000, B 0.000, C 0.000 }
gfCNCPoint4[669] = {X 13.9980, Y 38.1522, Z -4.6667, A 0.000, B 0.000, C 0.000 }
gfCNCPoint4[670] = {X 15.3127, Y 37.8963, Z -4.6667, A 0.000, B 0.000, C 0.000 }
gfCNCPoint4[671] = {X 16.5850, Y 37.4777, Z -4.6667, A 0.000, B 0.000, C 0.000 }
gfCNCPoint4[672] = {X 18.0105, Y 36.8099, Z -4.6667, A 0.000, B 0.000, C 0.000 }
gfCNCPoint4[673] = {X 19.3501, Y 35.9832, Z -4.6667, A 0.000, B 0.000, C 0.000 }
gfCNCPoint4[674] = {X 19.4352, Y 35.1814, Z -4.6667, A 0.000, B 0.000, C 0.000 }
gfCNCPoint4[675] = {X 19.6763, Y 34.4121, Z -4.6667, A 0.000, B 0.000, C 0.000 }
gfCNCPoint4[676] = {X 20.0640, Y 33.7052, Z -4.6667, A 0.000, B 0.000, C 0.000 }
gfCNCPoint4[677] = {X 18.0872, Y 34.0795, Z -4.6667, A 0.000, B 0.000, C 0.000 }
gfCNCPoint4[678] = {X 16.0874, Y 34.3004, Z -4.6667, A 0.000, B 0.000, C 0.000 }
gfCNCPoint4[679] = {X 15.3633, Y 34.3531, Z -4.6667, A 0.000, B 0.000, C 0.000 }
gfCNCPoint4[680] = {X 14.6391, Y 34.4036, Z -4.6667, A 0.000, B 0.000, C 0.000 }
gfCNCPoint4[681] = {X 10.6874, Y 35.0233, Z -4.6667, A 0.000, B 0.000, C 0.000 }
gfCNCPoint4[682] = {X 14.7701, Y 36.3192, Z -4.6667, A 0.000, B 0.000, C 0.000 }
gfCNCPoint4[683] = {X 14.6336, Y 34.3238, Z -4.6667, A 0.000, B 0.000, C 0.000 }
gfCNCPoint4[684] = {X 12.2421, Y 34.4759, Z -4.6667, A 0.000, B 0.000, C 0.000 }
gfCNCPoint4[685] = {X 9.8492, Y 34.6053, Z -4.6667, A 0.000, B 0.000, C 0.000 }
gfCNCPoint4[686] = {X 8.5937, Y 34.7142, Z -4.6667, A 0.000, B 0.000, C 0.000 }
gfCNCPoint4[687] = {X 7.3610, Y 34.9765, Z -4.6667, A 0.000, B 0.000, C 0.000 }
gfCNCPoint4[688] = {X 7.2802, Y 35.1979, Z -4.6667, A 0.000, B 0.000, C 0.000 }
gfCNCPoint4[689] = {X 7.2522, Y 35.4320, Z -4.6667, A 0.000, B 0.000, C 0.000 }
gfCNCPoint4[690] = {X 7.3216, Y 35.9825, Z -4.6667, A 0.000, B 0.000, C 0.000 }
gfCNCPoint4[691] = {X 7.5290, Y 36.4971, Z -4.6667, A 0.000, B 0.000, C 0.000 }
gfCNCPoint4[692] = {X 7.8607, Y 36.9418, Z -4.6667, A 0.000, B 0.000, C 0.000 }
gfCNCPoint4[693] = {X 8.2947, Y 37.2874, Z -4.6667, A 0.000, B 0.000, C 0.000 }
gfCNCPoint4[694] = {X 9.1153, Y 37.7037, Z -4.6667, A 0.000, B 0.000, C 0.000 }
gfCNCPoint4[695] = {X 9.9884, Y 37.9944, Z -4.6667, A 0.000, B 0.000, C 0.000 }
gfCNCPoint4[696] = {X 11.3149, Y 38.2420, Z -4.6667, A 0.000, B 0.000, C 0.000 }
gfCNCPoint4[697] = {X 12.6619, Y 38.3215, Z -4.6667, A 0.000, B 0.000, C 0.000 }
gfCNCPoint4[698] = {X 14.0084, Y 38.2316, Z -4.6667, A 0.000, B 0.000, C 0.000 }
gfCNCPoint4[699] = {X 15.3329, Y 37.9737, Z -4.6667, A 0.000, B 0.000, C 0.000 }
gfCNCPoint4[700] = {X 16.6147, Y 37.5520, Z -4.6667, A 0.000, B 0.000, C 0.000 }
gfCNCPoint4[701] = {X 18.0669, Y 36.8704, Z -4.6667, A 0.000, B 0.000, C 0.000 }
gfCNCPoint4[702] = {X 19.4300, Y 36.0248, Z -4.6667, A 0.000, B 0.000, C 0.000 }
gfCNCPoint4[703] = {X 19.5226, Y 35.1553, Z -4.6667, A 0.000, B 0.000, C 0.000 }
gfCNCPoint4[704] = {X 19.8019, Y 34.3266, Z -4.6667, A 0.000, B 0.000, C 0.000 }
gfCNCPoint4[705] = {X 20.2547, Y 33.5784, Z -4.6667, A 0.000, B 0.000, C 0.000 }
gfCNCPoint4[706] = {X 18.1812, Y 33.9843, Z -4.6667, A 0.000, B 0.000, C 0.000 }
gfCNCPoint4[707] = {X 16.0816, Y 34.2206, Z -4.6667, A 0.000, B 0.000, C 0.000 }
gfCNCPoint4[708] = {X 15.3577, Y 34.2733, Z -4.6667, A 0.000, B 0.000, C 0.000 }
gfCNCPoint4[709] = {X 14.6336, Y 34.3238, Z -4.6667, A 0.000, B 0.000, C 0.000 }
gfCNCPoint4[710] = {X 14.7701, Y 36.3192, Z -4.6667, A 0.000, B 0.000, C 0.000 }
gfCNCPoint4[711] = {X 14.7701, Y 36.3192, Z -1.6667, A 0.000, B 0.000, C 0.000 }
gfCNCPoint4[712] = {X 14.7701, Y 36.3192, Z 11.0000, A 0.000, B 0.000, C 0.000 }
gfCNCPoint4[713] = {X 15.0766, Y 19.4926, Z 11.0000, A 0.000, B 0.000, C 0.000 }
gfCNCPoint4[714] = {X 15.0766, Y 19.4926, Z -0.8333, A 0.000, B 0.000, C 0.000 }
gfCNCPoint4[715] = {X 14.5040, Y 19.3630, Z -0.9906, A 0.000, B 0.000, C 0.000 }
gfCNCPoint4[716] = {X 13.3045, Y 19.2494, Z -1.3135, A 0.000, B 0.000, C 0.000 }
gfCNCPoint4[717] = {X 12.0998, Y 19.2668, Z -1.6363, A 0.000, B 0.000, C 0.000 }
gfCNCPoint4[718] = {X 11.2937, Y 19.3825, Z -1.8545, A 0.000, B 0.000, C 0.000 }
gfCNCPoint4[719] = {X 10.6070, Y 19.4904, Z -2.0408, A 0.000, B 0.000, C 0.000 }
gfCNCPoint4[720] = {X 9.8990, Y 19.6134, Z -2.2333, A 0.000, B 0.000, C 0.000 }
gfCNCPoint4[721] = {X 8.6149, Y 20.0596, Z -2.5976, A 0.000, B 0.000, C 0.000 }
gfCNCPoint4[722] = {X 7.9833, Y 20.4021, Z -2.7901, A 0.000, B 0.000, C 0.000 }
gfCNCPoint4[723] = {X 7.9272, Y 20.9137, Z -2.9280, A 0.000, B 0.000, C 0.000 }
gfCNCPoint4[724] = {X 7.4493, Y 22.1322, Z -3.2787, A 0.000, B 0.000, C 0.000 }
gfCNCPoint4[725] = {X 7.1425, Y 22.5455, Z -3.4166, A 0.000, B 0.000, C 0.000 }
gfCNCPoint4[726] = {X 8.6596, Y 22.3485, Z -3.8266, A 0.000, B 0.000, C 0.000 }
gfCNCPoint4[727] = {X 8.9964, Y 22.3196, Z -3.9171, A 0.000, B 0.000, C 0.000 }
gfCNCPoint4[728] = {X 10.5268, Y 22.2552, Z -4.3275, A 0.000, B 0.000, C 0.000 }
gfCNCPoint4[729] = {X 11.1591, Y 22.2315, Z -4.4971, A 0.000, B 0.000, C 0.000 }
gfCNCPoint4[730] = {X 11.7913, Y 22.2024, Z -4.6667, A 0.000, B 0.000, C 0.000 }
gfCNCPoint4[731] = {X 14.1195, Y 22.0765, Z -4.6667, A 0.000, B 0.000, C 0.000 }
gfCNCPoint4[732] = {X 16.4455, Y 21.9134, Z -4.6667, A 0.000, B 0.000, C 0.000 }
gfCNCPoint4[733] = {X 17.0562, Y 21.8296, Z -4.6667, A 0.000, B 0.000, C 0.000 }
gfCNCPoint4[734] = {X 17.6529, Y 21.6751, Z -4.6667, A 0.000, B 0.000, C 0.000 }
gfCNCPoint4[735] = {X 17.6743, Y 21.2160, Z -4.6667, A 0.000, B 0.000, C 0.000 }
gfCNCPoint4[736] = {X 17.5245, Y 20.7816, Z -4.6667, A 0.000, B 0.000, C 0.000 }
gfCNCPoint4[737] = {X 17.2246, Y 20.4333, Z -4.6667, A 0.000, B 0.000, C 0.000 }
gfCNCPoint4[738] = {X 16.3055, Y 19.8928, Z -4.6667, A 0.000, B 0.000, C 0.000 }
gfCNCPoint4[739] = {X 15.2982, Y 19.5428, Z -4.6667, A 0.000, B 0.000, C 0.000 }
gfCNCPoint4[740] = {X 13.9732, Y 19.3266, Z -4.6667, A 0.000, B 0.000, C 0.000 }
gfCNCPoint4[741] = {X 12.6317, Y 19.2729, Z -4.6667, A 0.000, B 0.000, C 0.000 }
gfCNCPoint4[742] = {X 11.2937, Y 19.3825, Z -4.6667, A 0.000, B 0.000, C 0.000 }
gfCNCPoint4[743] = {X 10.6070, Y 19.4904, Z -4.6667, A 0.000, B 0.000, C 0.000 }
gfCNCPoint4[744] = {X 9.2580, Y 19.8395, Z -4.6667, A 0.000, B 0.000, C 0.000 }
gfCNCPoint4[745] = {X 7.9833, Y 20.4021, Z -4.6667, A 0.000, B 0.000, C 0.000 }
gfCNCPoint4[746] = {X 7.8312, Y 21.1626, Z -4.6667, A 0.000, B 0.000, C 0.000 }
gfCNCPoint4[747] = {X 7.5480, Y 21.8845, Z -4.6667, A 0.000, B 0.000, C 0.000 }
gfCNCPoint4[748] = {X 7.1425, Y 22.5455, Z -4.6667, A 0.000, B 0.000, C 0.000 }
gfCNCPoint4[749] = {X 8.8315, Y 22.3635, Z -4.6667, A 0.000, B 0.000, C 0.000 }
gfCNCPoint4[750] = {X 10.5268, Y 22.2552, Z -4.6667, A 0.000, B 0.000, C 0.000 }
gfCNCPoint4[751] = {X 11.1591, Y 22.2301, Z -4.6667, A 0.000, B 0.000, C 0.000 }
gfCNCPoint4[752] = {X 11.7913, Y 22.2024, Z -4.6667, A 0.000, B 0.000, C 0.000 }
gfCNCPoint4[753] = {X 7.7983, Y 22.1175, Z -4.6667, A 0.000, B 0.000, C 0.000 }
gfCNCPoint4[754] = {X 11.7949, Y 22.2823, Z -4.6667, A 0.000, B 0.000, C 0.000 }
gfCNCPoint4[755] = {X 14.1245, Y 22.1563, Z -4.6667, A 0.000, B 0.000, C 0.000 }
gfCNCPoint4[756] = {X 16.4517, Y 21.9932, Z -4.6667, A 0.000, B 0.000, C 0.000 }
gfCNCPoint4[757] = {X 17.0933, Y 21.9038, Z -4.6667, A 0.000, B 0.000, C 0.000 }
gfCNCPoint4[758] = {X 17.7194, Y 21.7376, Z -4.6667, A 0.000, B 0.000, C 0.000 }
gfCNCPoint4[759] = {X 17.7574, Y 21.2340, Z -4.6667, A 0.000, B 0.000, C 0.000 }
gfCNCPoint4[760] = {X 17.6008, Y 20.7539, Z -4.6667, A 0.000, B 0.000, C 0.000 }
gfCNCPoint4[761] = {X 17.2731, Y 20.3696, Z -4.6667, A 0.000, B 0.000, C 0.000 }
gfCNCPoint4[762] = {X 16.3395, Y 19.8204, Z -4.6667, A 0.000, B 0.000, C 0.000 }
gfCNCPoint4[763] = {X 15.3164, Y 19.4649, Z -4.6667, A 0.000, B 0.000, C 0.000 }
gfCNCPoint4[764] = {X 13.9814, Y 19.2471, Z -4.6667, A 0.000, B 0.000, C 0.000 }
gfCNCPoint4[765] = {X 12.6299, Y 19.1929, Z -4.6667, A 0.000, B 0.000, C 0.000 }
gfCNCPoint4[766] = {X 11.2818, Y 19.3034, Z -4.6667, A 0.000, B 0.000, C 0.000 }
gfCNCPoint4[767] = {X 10.5939, Y 19.4115, Z -4.6667, A 0.000, B 0.000, C 0.000 }
gfCNCPoint4[768] = {X 9.2121, Y 19.7708, Z -4.6667, A 0.000, B 0.000, C 0.000 }
gfCNCPoint4[769] = {X 7.9081, Y 20.3520, Z -4.6667, A 0.000, B 0.000, C 0.000 }
gfCNCPoint4[770] = {X 7.7440, Y 21.1752, Z -4.6667, A 0.000, B 0.000, C 0.000 }
gfCNCPoint4[771] = {X 7.4238, Y 21.9511, Z -4.6667, A 0.000, B 0.000, C 0.000 }
gfCNCPoint4[772] = {X 6.9596, Y 22.6504, Z -4.6667, A 0.000, B 0.000, C 0.000 }
gfCNCPoint4[773] = {X 8.7403, Y 22.4517, Z -4.6667, A 0.000, B 0.000, C 0.000 }
gfCNCPoint4[774] = {X 10.5282, Y 22.3352, Z -4.6667, A 0.000, B 0.000, C 0.000 }
gfCNCPoint4[775] = {X 11.1617, Y 22.3101, Z -4.6667, A 0.000, B 0.000, C 0.000 }
gfCNCPoint4[776] = {X 11.7949, Y 22.2823, Z -4.6667, A 0.000, B 0.000, C 0.000 }
gfCNCPoint4[777] = {X 15.7595, Y 21.7506, Z -4.6667, A 0.000, B 0.000, C 0.000 }
gfCNCPoint4[778] = {X 7.8020, Y 22.1974, Z -4.6667, A 0.000, B 0.000, C 0.000 }
gfCNCPoint4[779] = {X 11.7986, Y 22.3622, Z -4.6667, A 0.000, B 0.000, C 0.000 }
gfCNCPoint4[780] = {X 14.1294, Y 22.2362, Z -4.6667, A 0.000, B 0.000, C 0.000 }
gfCNCPoint4[781] = {X 16.4579, Y 22.0729, Z -4.6667, A 0.000, B 0.000, C 0.000 }
gfCNCPoint4[782] = {X 17.1297, Y 21.9780, Z -4.6667, A 0.000, B 0.000, C 0.000 }
gfCNCPoint4[783] = {X 17.7843, Y 21.8002, Z -4.6667, A 0.000, B 0.000, C 0.000 }
gfCNCPoint4[784] = {X 17.8399, Y 21.2523, Z -4.6667, A 0.000, B 0.000, C 0.000 }
gfCNCPoint4[785] = {X 17.6770, Y 20.7264, Z -4.6667, A 0.000, B 0.000, C 0.000 }
gfCNCPoint4[786] = {X 17.3215, Y 20.3059, Z -4.6667, A 0.000, B 0.000, C 0.000 }
gfCNCPoint4[787] = {X 16.3736, Y 19.7480, Z -4.6667, A 0.000, B 0.000, C 0.000 }
gfCNCPoint4[788] = {X 15.3346, Y 19.3870, Z -4.6667, A 0.000, B 0.000, C 0.000 }
gfCNCPoint4[789] = {X 13.9897, Y 19.1675, Z -4.6667, A 0.000, B 0.000, C 0.000 }
gfCNCPoint4[790] = {X 12.6280, Y 19.1130, Z -4.6667, A 0.000, B 0.000, C 0.000 }
gfCNCPoint4[791] = {X 11.2699, Y 19.2243, Z -4.6667, A 0.000, B 0.000, C 0.000 }
gfCNCPoint4[792] = {X 10.5809, Y 19.3326, Z -4.6667, A 0.000, B 0.000, C 0.000 }
gfCNCPoint4[793] = {X 9.6302, Y 19.5528, Z -4.6667, A 0.000, B 0.000, C 0.000 }
gfCNCPoint4[794] = {X 8.7100, Y 19.8776, Z -4.6667, A 0.000, B 0.000, C 0.000 }
gfCNCPoint4[795] = {X 7.8317, Y 20.3028, Z -4.6667, A 0.000, B 0.000, C 0.000 }
gfCNCPoint4[796] = {X 7.8285, Y 20.3441, Z -4.6667, A 0.000, B 0.000, C 0.000 }
gfCNCPoint4[797] = {X 7.6467, Y 21.2184, Z -4.6667, A 0.000, B 0.000, C 0.000 }
gfCNCPoint4[798] = {X 7.2859, Y 22.0352, Z -4.6667, A 0.000, B 0.000, C 0.000 }
gfCNCPoint4[799] = {X 6.7619, Y 22.7584, Z -4.6667, A 0.000, B 0.000, C 0.000 }
gfCNCPoint4[800] = {X 8.6426, Y 22.5408, Z -4.6667, A 0.000, B 0.000, C 0.000 }
gfCNCPoint4[801] = {X 10.5316, Y 22.4151, Z -4.6667, A 0.000, B 0.000, C 0.000 }
gfCNCPoint4[802] = {X 11.1652, Y 22.3900, Z -4.6667, A 0.000, B 0.000, C 0.000 }
gfCNCPoint4[803] = {X 11.7986, Y 22.3622, Z -4.6667, A 0.000, B 0.000, C 0.000 }
gfCNCPoint4[804] = {X 15.7631, Y 21.8305, Z -4.6667, A 0.000, B 0.000, C 0.000 }
gfCNCPoint4[805] = {X 7.8057, Y 22.2773, Z -4.6667, A 0.000, B 0.000, C 0.000 }
gfCNCPoint4[806] = {X 11.8023, Y 22.4421, Z -4.6667, A 0.000, B 0.000, C 0.000 }
gfCNCPoint4[807] = {X 14.1344, Y 22.3160, Z -4.6667, A 0.000, B 0.000, C 0.000 }
gfCNCPoint4[808] = {X 16.4641, Y 22.1527, Z -4.6667, A 0.000, B 0.000, C 0.000 }
gfCNCPoint4[809] = {X 17.1654, Y 22.0523, Z -4.6667, A 0.000, B 0.000, C 0.000 }
gfCNCPoint4[810] = {X 17.8480, Y 21.8629, Z -4.6667, A 0.000, B 0.000, C 0.000 }
gfCNCPoint4[811] = {X 17.9264, Y 21.4211, Z -4.6667, A 0.000, B 0.000, C 0.000 }
gfCNCPoint4[812] = {X 17.8670, Y 20.9764, Z -4.6667, A 0.000, B 0.000, C 0.000 }
gfCNCPoint4[813] = {X 17.6755, Y 20.5706, Z -4.6667, A 0.000, B 0.000, C 0.000 }
gfCNCPoint4[814] = {X 17.3699, Y 20.2422, Z -4.6667, A 0.000, B 0.000, C 0.000 }
gfCNCPoint4[815] = {X 16.4076, Y 19.6756, Z -4.6667, A 0.000, B 0.000, C 0.000 }
gfCNCPoint4[816] = {X 15.3528, Y 19.3091, Z -4.6667, A 0.000, B 0.000, C 0.000 }
gfCNCPoint4[817] = {X 13.9979, Y 19.0879, Z -4.6667, A 0.000, B 0.000, C 0.000 }
gfCNCPoint4[818] = {X 12.6262, Y 19.0330, Z -4.6667, A 0.000, B 0.000, C 0.000 }
gfCNCPoint4[819] = {X 11.2580, Y 19.1451, Z -4.6667, A 0.000, B 0.000, C 0.000 }
gfCNCPoint4[820] = {X 10.5678, Y 19.2536, Z -4.6667, A 0.000, B 0.000, C 0.000 }
gfCNCPoint4[821] = {X 9.5944, Y 19.4799, Z -4.6667, A 0.000, B 0.000, C 0.000 }
gfCNCPoint4[822] = {X 8.6529, Y 19.8148, Z -4.6667, A 0.000, B 0.000, C 0.000 }
gfCNCPoint4[823] = {X 7.7552, Y 20.2539, Z -4.6667, A 0.000, B 0.000, C 0.000 }
gfCNCPoint4[824] = {X 7.7492, Y 20.3322, Z -4.6667, A 0.000, B 0.000, C 0.000 }
gfCNCPoint4[825] = {X 7.5475, Y 21.2637, Z -4.6667, A 0.000, B 0.000, C 0.000 }
gfCNCPoint4[826] = {X 7.1390, Y 22.1248, Z -4.6667, A 0.000, B 0.000, C 0.000 }
gfCNCPoint4[827] = {X 6.5453, Y 22.8703, Z -4.6667, A 0.000, B 0.000, C 0.000 }
gfCNCPoint4[828] = {X 8.5353, Y 22.6311, Z -4.6667, A 0.000, B 0.000, C 0.000 }
gfCNCPoint4[829] = {X 10.5350, Y 22.4950, Z -4.6667, A 0.000, B 0.000, C 0.000 }
gfCNCPoint4[830] = {X 11.1687, Y 22.4699, Z -4.6667, A 0.000, B 0.000, C 0.000 }
gfCNCPoint4[831] = {X 11.8023, Y 22.4421, Z -4.6667, A 0.000, B 0.000, C 0.000 }
gfCNCPoint4[832] = {X 15.7668, Y 21.9104, Z -4.6667, A 0.000, B 0.000, C 0.000 }
gfCNCPoint4[833] = {X 7.8094, Y 22.3572, Z -4.6667, A 0.000, B 0.000, C 0.000 }
gfCNCPoint4[834] = {X 11.8060, Y 22.5220, Z -4.6667, A 0.000, B 0.000, C 0.000 }
gfCNCPoint4[835] = {X 14.1393, Y 22.3958, Z -4.6667, A 0.000, B 0.000, C 0.000 }
gfCNCPoint4[836] = {X 16.4704, Y 22.2324, Z -4.6667, A 0.000, B 0.000, C 0.000 }
gfCNCPoint4[837] = {X 17.2006, Y 22.1266, Z -4.6667, A 0.000, B 0.000, C 0.000 }
gfCNCPoint4[838] = {X 17.9105, Y 21.9257, Z -4.6667, A 0.000, B 0.000, C 0.000 }
gfCNCPoint4[839] = {X 18.0055, Y 21.4518, Z -4.6667, A 0.000, B 0.000, C 0.000 }
gfCNCPoint4[840] = {X 17.9490, Y 20.9718, Z -4.6667, A 0.000, B 0.000, C 0.000 }
gfCNCPoint4[841] = {X 17.7466, Y 20.5330, Z -4.6667, A 0.000, B 0.000, C 0.000 }
gfCNCPoint4[842] = {X 17.4182, Y 20.1784, Z -4.6667, A 0.000, B 0.000, C 0.000 }
gfCNCPoint4[843] = {X 16.4416, Y 19.6032, Z -4.6667, A 0.000, B 0.000, C 0.000 }
gfCNCPoint4[844] = {X 15.3709, Y 19.2312, Z -4.6667, A 0.000, B 0.000, C 0.000 }
gfCNCPoint4[845] = {X 14.0061, Y 19.0083, Z -4.6667, A 0.000, B 0.000, C 0.000 }
gfCNCPoint4[846] = {X 12.6243, Y 18.9530, Z -4.6667, A 0.000, B 0.000, C 0.000 }
gfCNCPoint4[847] = {X 11.2461, Y 19.0660, Z -4.6667, A 0.000, B 0.000, C 0.000 }
gfCNCPoint4[848] = {X 10.5547, Y 19.1747, Z -4.6667, A 0.000, B 0.000, C 0.000 }
gfCNCPoint4[849] = {X 9.5586, Y 19.4071, Z -4.6667, A 0.000, B 0.000, C 0.000 }
gfCNCPoint4[850] = {X 8.5957, Y 19.7521, Z -4.6667, A 0.000, B 0.000, C 0.000 }
gfCNCPoint4[851] = {X 7.6787, Y 20.2052, Z -4.6667, A 0.000, B 0.000, C 0.000 }
gfCNCPoint4[852] = {X 7.6695, Y 20.3253, Z -4.6667, A 0.000, B 0.000, C 0.000 }
gfCNCPoint4[853] = {X 7.5231, Y 21.0760, Z -4.6667, A 0.000, B 0.000, C 0.000 }
gfCNCPoint4[854] = {X 7.2392, Y 21.7862, Z -4.6667, A 0.000, B 0.000, C 0.000 }
gfCNCPoint4[855] = {X 6.8276, Y 22.4310, Z -4.6667, A 0.000, B 0.000, C 0.000 }
gfCNCPoint4[856] = {X 6.3030, Y 22.9875, Z -4.6667, A 0.000, B 0.000, C 0.000 }
gfCNCPoint4[857] = {X 8.4150, Y 22.7229, Z -4.6667, A 0.000, B 0.000, C 0.000 }
gfCNCPoint4[858] = {X 10.5383, Y 22.5749, Z -4.6667, A 0.000, B 0.000, C 0.000 }
gfCNCPoint4[859] = {X 11.1722, Y 22.5499, Z -4.6667, A 0.000, B 0.000, C 0.000 }
gfCNCPoint4[860] = {X 11.8060, Y 22.5220, Z -4.6667, A 0.000, B 0.000, C 0.000 }
gfCNCPoint4[861] = {X 15.7705, Y 21.9904, Z -4.6667, A 0.000, B 0.000, C 0.000 }
gfCNCPoint4[862] = {X 11.7347, Y 22.6054, Z -4.6667, A 0.000, B 0.000, C 0.000 }
gfCNCPoint4[863] = {X 11.8097, Y 22.6019, Z -4.6667, A 0.000, B 0.000, C 0.000 }
gfCNCPoint4[864] = {X 14.1443, Y 22.4757, Z -4.6667, A 0.000, B 0.000, C 0.000 }
gfCNCPoint4[865] = {X 16.4766, Y 22.3122, Z -4.6667, A 0.000, B 0.000, C 0.000 }
gfCNCPoint4[866] = {X 17.2353, Y 22.2010, Z -4.6667, A 0.000, B 0.000, C 0.000 }
gfCNCPoint4[867] = {X 17.9721, Y 21.9886, Z -4.6667, A 0.000, B 0.000, C 0.000 }
gfCNCPoint4[868] = {X 18.0841, Y 21.4828, Z -4.6667, A 0.000, B 0.000, C 0.000 }
gfCNCPoint4[869] = {X 18.0308, Y 20.9676, Z -4.6667, A 0.000, B 0.000, C 0.000 }
gfCNCPoint4[870] = {X 17.8177, Y 20.4954, Z -4.6667, A 0.000, B 0.000, C 0.000 }
gfCNCPoint4[871] = {X 17.4665, Y 20.1146, Z -4.6667, A 0.000, B 0.000, C 0.000 }
gfCNCPoint4[872] = {X 16.4756, Y 19.5307, Z -4.6667, A 0.000, B 0.000, C 0.000 }
gfCNCPoint4[873] = {X 15.3891, Y 19.1532, Z -4.6667, A 0.000, B 0.000, C 0.000 }
gfCNCPoint4[874] = {X 14.0143, Y 18.9287, Z -4.6667, A 0.000, B 0.000, C 0.000 }
gfCNCPoint4[875] = {X 12.6225, Y 18.8730, Z -4.6667, A 0.000, B 0.000, C 0.000 }
gfCNCPoint4[876] = {X 11.2342, Y 18.9869, Z -4.6667, A 0.000, B 0.000, C 0.000 }
gfCNCPoint4[877] = {X 10.5417, Y 19.0958, Z -4.6667, A 0.000, B 0.000, C 0.000 }
gfCNCPoint4[878] = {X 9.5228, Y 19.3343, Z -4.6667, A 0.000, B 0.000, C 0.000 }
gfCNCPoint4[879] = {X 8.5385, Y 19.6895, Z -4.6667, A 0.000, B 0.000, C 0.000 }
gfCNCPoint4[880] = {X 7.6021, Y 20.1568, Z -4.6667, A 0.000, B 0.000, C 0.000 }
gfCNCPoint4[881] = {X 7.5898, Y 20.3183, Z -4.6667, A 0.000, B 0.000, C 0.000 }
gfCNCPoint4[882] = {X 7.4462, Y 21.0541, Z -4.6667, A 0.000, B 0.000, C 0.000 }
gfCNCPoint4[883] = {X 7.1678, Y 21.7501, Z -4.6667, A 0.000, B 0.000, C 0.000 }
gfCNCPoint4[884] = {X 6.7644, Y 22.3820, Z -4.6667, A 0.000, B 0.000, C 0.000 }
gfCNCPoint4[885] = {X 6.2502, Y 22.9275, Z -4.6667, A 0.000, B 0.000, C 0.000 }
gfCNCPoint4[886] = {X 6.2082, Y 22.9638, Z -4.6667, A 0.000, B 0.000, C 0.000 }
gfCNCPoint4[887] = {X 6.1658, Y 22.9996, Z -4.6667, A 0.000, B 0.000, C 0.000 }
gfCNCPoint4[888] = {X 6.1508, Y 23.0922, Z -4.6667, A 0.000, B 0.000, C 0.000 }
gfCNCPoint4[889] = {X 6.2329, Y 23.0793, Z -4.6667, A 0.000, B 0.000, C 0.000 }
gfCNCPoint4[890] = {X 6.3151, Y 23.0666, Z -4.6667, A 0.000, B 0.000, C 0.000 }
gfCNCPoint4[891] = {X 8.4227, Y 22.8026, Z -4.6667, A 0.000, B 0.000, C 0.000 }
gfCNCPoint4[892] = {X 10.5417, Y 22.6549, Z -4.6667, A 0.000, B 0.000, C 0.000 }
gfCNCPoint4[893] = {X 11.1757, Y 22.6298, Z -4.6667, A 0.000, B 0.000, C 0.000 }
gfCNCPoint4[894] = {X 11.8097, Y 22.6019, Z -4.6667, A 0.000, B 0.000, C 0.000 }
gfCNCPoint4[895] = {X 11.7176, Y 20.6041, Z -4.6667, A 0.000, B 0.000, C 0.000 }
gfCNCPoint4[896] = {X 11.7176, Y 20.6041, Z -1.6667, A 0.000, B 0.000, C 0.000 }
gfCNCPoint4[897] = {X 11.7176, Y 20.6041, Z 11.0000, A 0.000, B 0.000, C 0.000 }
gfCNCPoint4[898] = {X 15.0773, Y 19.4931, Z 11.0000, A 0.000, B 0.000, C 0.000 }
gfCNCPoint4[899] = {X 15.0773, Y 19.4931, Z -1.6667, A 0.000, B 0.000, C 0.000 }
gfCNCPoint4[900] = {X 14.5040, Y 19.3634, Z -1.8242, A 0.000, B 0.000, C 0.000 }
gfCNCPoint4[901] = {X 13.3045, Y 19.2497, Z -2.1470, A 0.000, B 0.000, C 0.000 }
gfCNCPoint4[902] = {X 12.0998, Y 19.2671, Z -2.4699, A 0.000, B 0.000, C 0.000 }
gfCNCPoint4[903] = {X 11.2937, Y 19.3828, Z -2.6881, A 0.000, B 0.000, C 0.000 }
gfCNCPoint4[904] = {X 10.6070, Y 19.4908, Z -2.8743, A 0.000, B 0.000, C 0.000 }
gfCNCPoint4[905] = {X 9.8991, Y 19.6137, Z -3.0668, A 0.000, B 0.000, C 0.000 }
gfCNCPoint4[906] = {X 8.6148, Y 20.0600, Z -3.4312, A 0.000, B 0.000, C 0.000 }
gfCNCPoint4[907] = {X 7.9832, Y 20.4025, Z -3.6237, A 0.000, B 0.000, C 0.000 }
gfCNCPoint4[908] = {X 7.9271, Y 20.9141, Z -3.7616, A 0.000, B 0.000, C 0.000 }
gfCNCPoint4[909] = {X 7.4494, Y 22.1320, Z -4.1121, A 0.000, B 0.000, C 0.000 }
gfCNCPoint4[910] = {X 7.1427, Y 22.5453, Z -4.2500, A 0.000, B 0.000, C 0.000 }
gfCNCPoint4[911] = {X 8.6614, Y 22.3481, Z -4.6604, A 0.000, B 0.000, C 0.000 }
gfCNCPoint4[912] = {X 8.9947, Y 22.3195, Z -4.7500, A 0.000, B 0.000, C 0.000 }
gfCNCPoint4[913] = {X 10.5268, Y 22.2548, Z -5.1609, A 0.000, B 0.000, C 0.000 }
gfCNCPoint4[914] = {X 11.1591, Y 22.2312, Z -5.3304, A 0.000, B 0.000, C 0.000 }
gfCNCPoint4[915] = {X 11.7913, Y 22.2020, Z -5.5000, A 0.000, B 0.000, C 0.000 }
gfCNCPoint4[916] = {X 14.1195, Y 22.0761, Z -5.5000, A 0.000, B 0.000, C 0.000 }
gfCNCPoint4[917] = {X 16.4453, Y 21.9131, Z -5.5000, A 0.000, B 0.000, C 0.000 }
gfCNCPoint4[918] = {X 17.0559, Y 21.8293, Z -5.5000, A 0.000, B 0.000, C 0.000 }
gfCNCPoint4[919] = {X 17.6526, Y 21.6749, Z -5.5000, A 0.000, B 0.000, C 0.000 }
gfCNCPoint4[920] = {X 17.6740, Y 21.2160, Z -5.5000, A 0.000, B 0.000, C 0.000 }
gfCNCPoint4[921] = {X 17.5242, Y 20.7818, Z -5.5000, A 0.000, B 0.000, C 0.000 }
gfCNCPoint4[922] = {X 17.2246, Y 20.4336, Z -5.5000, A 0.000, B 0.000, C 0.000 }
gfCNCPoint4[923] = {X 16.3055, Y 19.8931, Z -5.5000, A 0.000, B 0.000, C 0.000 }
gfCNCPoint4[924] = {X 15.2982, Y 19.5431, Z -5.5000, A 0.000, B 0.000, C 0.000 }
gfCNCPoint4[925] = {X 13.9732, Y 19.3270, Z -5.5000, A 0.000, B 0.000, C 0.000 }
gfCNCPoint4[926] = {X 12.6317, Y 19.2733, Z -5.5000, A 0.000, B 0.000, C 0.000 }
gfCNCPoint4[927] = {X 11.2937, Y 19.3828, Z -5.5000, A 0.000, B 0.000, C 0.000 }
gfCNCPoint4[928] = {X 10.6070, Y 19.4908, Z -5.5000, A 0.000, B 0.000, C 0.000 }
gfCNCPoint4[929] = {X 9.2580, Y 19.8398, Z -5.5000, A 0.000, B 0.000, C 0.000 }
gfCNCPoint4[930] = {X 7.9832, Y 20.4025, Z -5.5000, A 0.000, B 0.000, C 0.000 }
gfCNCPoint4[931] = {X 7.8312, Y 21.1627, Z -5.5000, A 0.000, B 0.000, C 0.000 }
gfCNCPoint4[932] = {X 7.5481, Y 21.8844, Z -5.5000, A 0.000, B 0.000, C 0.000 }
gfCNCPoint4[933] = {X 7.1427, Y 22.5453, Z -5.5000, A 0.000, B 0.000, C 0.000 }
gfCNCPoint4[934] = {X 8.8316, Y 22.3633, Z -5.5000, A 0.000, B 0.000, C 0.000 }
gfCNCPoint4[935] = {X 10.5268, Y 22.2548, Z -5.5000, A 0.000, B 0.000, C 0.000 }
gfCNCPoint4[936] = {X 11.1591, Y 22.2298, Z -5.5000, A 0.000, B 0.000, C 0.000 }
gfCNCPoint4[937] = {X 11.7913, Y 22.2020, Z -5.5000, A 0.000, B 0.000, C 0.000 }
gfCNCPoint4[938] = {X 7.7984, Y 22.1171, Z -5.5000, A 0.000, B 0.000, C 0.000 }
gfCNCPoint4[939] = {X 11.7950, Y 22.2820, Z -5.5000, A 0.000, B 0.000, C 0.000 }
gfCNCPoint4[940] = {X 14.1244, Y 22.1560, Z -5.5000, A 0.000, B 0.000, C 0.000 }
gfCNCPoint4[941] = {X 16.4516, Y 21.9928, Z -5.5000, A 0.000, B 0.000, C 0.000 }
gfCNCPoint4[942] = {X 17.0931, Y 21.9035, Z -5.5000, A 0.000, B 0.000, C 0.000 }
gfCNCPoint4[943] = {X 17.7191, Y 21.7373, Z -5.5000, A 0.000, B 0.000, C 0.000 }
gfCNCPoint4[944] = {X 17.7571, Y 21.2340, Z -5.5000, A 0.000, B 0.000, C 0.000 }
gfCNCPoint4[945] = {X 17.6005, Y 20.7541, Z -5.5000, A 0.000, B 0.000, C 0.000 }
gfCNCPoint4[946] = {X 17.2730, Y 20.3699, Z -5.5000, A 0.000, B 0.000, C 0.000 }
gfCNCPoint4[947] = {X 16.3395, Y 19.8207, Z -5.5000, A 0.000, B 0.000, C 0.000 }
gfCNCPoint4[948] = {X 15.3164, Y 19.4652, Z -5.5000, A 0.000, B 0.000, C 0.000 }
gfCNCPoint4[949] = {X 13.9814, Y 19.2474, Z -5.5000, A 0.000, B 0.000, C 0.000 }
gfCNCPoint4[950] = {X 12.6299, Y 19.1933, Z -5.5000, A 0.000, B 0.000, C 0.000 }
gfCNCPoint4[951] = {X 11.2818, Y 19.3037, Z -5.5000, A 0.000, B 0.000, C 0.000 }
gfCNCPoint4[952] = {X 10.5939, Y 19.4118, Z -5.5000, A 0.000, B 0.000, C 0.000 }
gfCNCPoint4[953] = {X 9.2116, Y 19.7713, Z -5.5000, A 0.000, B 0.000, C 0.000 }
gfCNCPoint4[954] = {X 7.9071, Y 20.3529, Z -5.5000, A 0.000, B 0.000, C 0.000 }
gfCNCPoint4[955] = {X 7.7432, Y 21.1756, Z -5.5000, A 0.000, B 0.000, C 0.000 }
gfCNCPoint4[956] = {X 7.4233, Y 21.9511, Z -5.5000, A 0.000, B 0.000, C 0.000 }
gfCNCPoint4[957] = {X 6.9596, Y 22.6502, Z -5.5000, A 0.000, B 0.000, C 0.000 }
gfCNCPoint4[958] = {X 8.7403, Y 22.4515, Z -5.5000, A 0.000, B 0.000, C 0.000 }
gfCNCPoint4[959] = {X 10.5282, Y 22.3348, Z -5.5000, A 0.000, B 0.000, C 0.000 }
gfCNCPoint4[960] = {X 11.1616, Y 22.3098, Z -5.5000, A 0.000, B 0.000, C 0.000 }
gfCNCPoint4[961] = {X 11.7950, Y 22.2820, Z -5.5000, A 0.000, B 0.000, C 0.000 }
gfCNCPoint4[962] = {X 15.7595, Y 21.7503, Z -5.5000, A 0.000, B 0.000, C 0.000 }
gfCNCPoint4[963] = {X 7.8020, Y 22.1970, Z -5.5000, A 0.000, B 0.000, C 0.000 }
gfCNCPoint4[964] = {X 11.7986, Y 22.3619, Z -5.5000, A 0.000, B 0.000, C 0.000 }
gfCNCPoint4[965] = {X 14.1294, Y 22.2358, Z -5.5000, A 0.000, B 0.000, C 0.000 }
gfCNCPoint4[966] = {X 16.4578, Y 22.0726, Z -5.5000, A 0.000, B 0.000, C 0.000 }
gfCNCPoint4[967] = {X 17.1294, Y 21.9777, Z -5.5000, A 0.000, B 0.000, C 0.000 }
gfCNCPoint4[968] = {X 17.7841, Y 21.7999, Z -5.5000, A 0.000, B 0.000, C 0.000 }
gfCNCPoint4[969] = {X 17.8396, Y 21.2523, Z -5.5000, A 0.000, B 0.000, C 0.000 }
gfCNCPoint4[970] = {X 17.6767, Y 20.7266, Z -5.5000, A 0.000, B 0.000, C 0.000 }
gfCNCPoint4[971] = {X 17.3214, Y 20.3062, Z -5.5000, A 0.000, B 0.000, C 0.000 }
gfCNCPoint4[972] = {X 16.3736, Y 19.7483, Z -5.5000, A 0.000, B 0.000, C 0.000 }
gfCNCPoint4[973] = {X 15.3346, Y 19.3873, Z -5.5000, A 0.000, B 0.000, C 0.000 }
gfCNCPoint4[974] = {X 13.9897, Y 19.1678, Z -5.5000, A 0.000, B 0.000, C 0.000 }
gfCNCPoint4[975] = {X 12.6280, Y 19.1133, Z -5.5000, A 0.000, B 0.000, C 0.000 }
gfCNCPoint4[976] = {X 11.2699, Y 19.2246, Z -5.5000, A 0.000, B 0.000, C 0.000 }
gfCNCPoint4[977] = {X 10.5808, Y 19.3329, Z -5.5000, A 0.000, B 0.000, C 0.000 }
gfCNCPoint4[978] = {X 9.6301, Y 19.5532, Z -5.5000, A 0.000, B 0.000, C 0.000 }
gfCNCPoint4[979] = {X 8.7098, Y 19.8780, Z -5.5000, A 0.000, B 0.000, C 0.000 }
gfCNCPoint4[980] = {X 7.8314, Y 20.3032, Z -5.5000, A 0.000, B 0.000, C 0.000 }
gfCNCPoint4[981] = {X 7.6544, Y 21.1921, Z -5.5000, A 0.000, B 0.000, C 0.000 }
gfCNCPoint4[982] = {X 7.2924, Y 22.0231, Z -5.5000, A 0.000, B 0.000, C 0.000 }
gfCNCPoint4[983] = {X 6.7621, Y 22.7581, Z -5.5000, A 0.000, B 0.000, C 0.000 }
gfCNCPoint4[984] = {X 8.6427, Y 22.5406, Z -5.5000, A 0.000, B 0.000, C 0.000 }
gfCNCPoint4[985] = {X 10.5316, Y 22.4148, Z -5.5000, A 0.000, B 0.000, C 0.000 }
gfCNCPoint4[986] = {X 11.1652, Y 22.3897, Z -5.5000, A 0.000, B 0.000, C 0.000 }
gfCNCPoint4[987] = {X 11.7986, Y 22.3619, Z -5.5000, A 0.000, B 0.000, C 0.000 }
gfCNCPoint4[988] = {X 15.7632, Y 21.8302, Z -5.5000, A 0.000, B 0.000, C 0.000 }
gfCNCPoint4[989] = {X 7.8057, Y 22.2770, Z -5.5000, A 0.000, B 0.000, C 0.000 }
gfCNCPoint4[990] = {X 11.8023, Y 22.4418, Z -5.5000, A 0.000, B 0.000, C 0.000 }
gfCNCPoint4[991] = {X 14.1343, Y 22.3157, Z -5.5000, A 0.000, B 0.000, C 0.000 }
gfCNCPoint4[992] = {X 16.4640, Y 22.1524, Z -5.5000, A 0.000, B 0.000, C 0.000 }
gfCNCPoint4[993] = {X 17.1652, Y 22.0520, Z -5.5000, A 0.000, B 0.000, C 0.000 }
gfCNCPoint4[994] = {X 17.8477, Y 21.8626, Z -5.5000, A 0.000, B 0.000, C 0.000 }
gfCNCPoint4[995] = {X 17.9261, Y 21.4210, Z -5.5000, A 0.000, B 0.000, C 0.000 }
gfCNCPoint4[996] = {X 17.8667, Y 20.9765, Z -5.5000, A 0.000, B 0.000, C 0.000 }
gfCNCPoint4[997] = {X 17.6753, Y 20.5709, Z -5.5000, A 0.000, B 0.000, C 0.000 }
gfCNCPoint4[998] = {X 17.3698, Y 20.2425, Z -5.5000, A 0.000, B 0.000, C 0.000 }
gfCNCPoint4[999] = {X 16.4076, Y 19.6759, Z -5.5000, A 0.000, B 0.000, C 0.000 }
gfCNCPoint4[1000] = {X 15.3528, Y 19.3094, Z -5.5000, A 0.000, B 0.000, C 0.000 }
gfCNCPoint4[1001] = {X 13.9979, Y 19.0882, Z -5.5000, A 0.000, B 0.000, C 0.000 }
gfCNCPoint4[1002] = {X 12.6262, Y 19.0333, Z -5.5000, A 0.000, B 0.000, C 0.000 }
gfCNCPoint4[1003] = {X 11.2580, Y 19.1455, Z -5.5000, A 0.000, B 0.000, C 0.000 }
gfCNCPoint4[1004] = {X 10.5678, Y 19.2540, Z -5.5000, A 0.000, B 0.000, C 0.000 }
gfCNCPoint4[1005] = {X 9.5945, Y 19.4802, Z -5.5000, A 0.000, B 0.000, C 0.000 }
gfCNCPoint4[1006] = {X 8.6530, Y 19.8150, Z -5.5000, A 0.000, B 0.000, C 0.000 }
gfCNCPoint4[1007] = {X 7.7553, Y 20.2541, Z -5.5000, A 0.000, B 0.000, C 0.000 }
gfCNCPoint4[1008] = {X 7.5634, Y 21.2139, Z -5.5000, A 0.000, B 0.000, C 0.000 }
gfCNCPoint4[1009] = {X 7.1526, Y 22.1022, Z -5.5000, A 0.000, B 0.000, C 0.000 }
gfCNCPoint4[1010] = {X 6.5456, Y 22.8700, Z -5.5000, A 0.000, B 0.000, C 0.000 }
gfCNCPoint4[1011] = {X 8.5354, Y 22.6309, Z -5.5000, A 0.000, B 0.000, C 0.000 }
gfCNCPoint4[1012] = {X 10.5350, Y 22.4947, Z -5.5000, A 0.000, B 0.000, C 0.000 }
gfCNCPoint4[1013] = {X 11.1687, Y 22.4696, Z -5.5000, A 0.000, B 0.000, C 0.000 }
gfCNCPoint4[1014] = {X 11.8023, Y 22.4418, Z -5.5000, A 0.000, B 0.000, C 0.000 }
gfCNCPoint4[1015] = {X 15.7668, Y 21.9101, Z -5.5000, A 0.000, B 0.000, C 0.000 }
gfCNCPoint4[1016] = {X 7.8094, Y 22.3569, Z -5.5000, A 0.000, B 0.000, C 0.000 }
gfCNCPoint4[1017] = {X 11.8060, Y 22.5217, Z -5.5000, A 0.000, B 0.000, C 0.000 }
gfCNCPoint4[1018] = {X 14.1393, Y 22.3955, Z -5.5000, A 0.000, B 0.000, C 0.000 }
gfCNCPoint4[1019] = {X 16.4702, Y 22.2321, Z -5.5000, A 0.000, B 0.000, C 0.000 }
gfCNCPoint4[1020] = {X 17.2004, Y 22.1263, Z -5.5000, A 0.000, B 0.000, C 0.000 }
gfCNCPoint4[1021] = {X 17.9103, Y 21.9254, Z -5.5000, A 0.000, B 0.000, C 0.000 }
gfCNCPoint4[1022] = {X 18.0052, Y 21.4517, Z -5.5000, A 0.000, B 0.000, C 0.000 }
gfCNCPoint4[1023] = {X 17.9487, Y 20.9720, Z -5.5000, A 0.000, B 0.000, C 0.000 }
gfCNCPoint4[1024] = {X 17.7464, Y 20.5332, Z -5.5000, A 0.000, B 0.000, C 0.000 }
gfCNCPoint4[1025] = {X 17.4182, Y 20.1787, Z -5.5000, A 0.000, B 0.000, C 0.000 }
gfCNCPoint4[1026] = {X 16.4416, Y 19.6034, Z -5.5000, A 0.000, B 0.000, C 0.000 }
gfCNCPoint4[1027] = {X 15.3709, Y 19.2315, Z -5.5000, A 0.000, B 0.000, C 0.000 }
gfCNCPoint4[1028] = {X 14.0061, Y 19.0087, Z -5.5000, A 0.000, B 0.000, C 0.000 }
gfCNCPoint4[1029] = {X 12.6243, Y 18.9533, Z -5.5000, A 0.000, B 0.000, C 0.000 }
gfCNCPoint4[1030] = {X 11.2461, Y 19.0664, Z -5.5000, A 0.000, B 0.000, C 0.000 }
gfCNCPoint4[1031] = {X 10.5547, Y 19.1750, Z -5.5000, A 0.000, B 0.000, C 0.000 }
gfCNCPoint4[1032] = {X 9.5587, Y 19.4074, Z -5.5000, A 0.000, B 0.000, C 0.000 }
gfCNCPoint4[1033] = {X 8.5958, Y 19.7523, Z -5.5000, A 0.000, B 0.000, C 0.000 }
gfCNCPoint4[1034] = {X 7.6789, Y 20.2054, Z -5.5000, A 0.000, B 0.000, C 0.000 }
gfCNCPoint4[1035] = {X 7.6695, Y 20.3253, Z -5.5000, A 0.000, B 0.000, C 0.000 }
gfCNCPoint4[1036] = {X 7.5231, Y 21.0759, Z -5.5000, A 0.000, B 0.000, C 0.000 }
gfCNCPoint4[1037] = {X 7.2393, Y 21.7860, Z -5.5000, A 0.000, B 0.000, C 0.000 }
gfCNCPoint4[1038] = {X 6.8279, Y 22.4307, Z -5.5000, A 0.000, B 0.000, C 0.000 }
gfCNCPoint4[1039] = {X 6.3034, Y 22.9872, Z -5.5000, A 0.000, B 0.000, C 0.000 }
gfCNCPoint4[1040] = {X 8.4152, Y 22.7227, Z -5.5000, A 0.000, B 0.000, C 0.000 }
gfCNCPoint4[1041] = {X 10.5383, Y 22.5746, Z -5.5000, A 0.000, B 0.000, C 0.000 }
gfCNCPoint4[1042] = {X 11.1722, Y 22.5495, Z -5.5000, A 0.000, B 0.000, C 0.000 }
gfCNCPoint4[1043] = {X 11.8060, Y 22.5217, Z -5.5000, A 0.000, B 0.000, C 0.000 }
gfCNCPoint4[1044] = {X 15.7705, Y 21.9900, Z -5.5000, A 0.000, B 0.000, C 0.000 }
gfCNCPoint4[1045] = {X 11.7347, Y 22.6051, Z -5.5000, A 0.000, B 0.000, C 0.000 }
gfCNCPoint4[1046] = {X 11.8097, Y 22.6016, Z -5.5000, A 0.000, B 0.000, C 0.000 }
gfCNCPoint4[1047] = {X 14.1442, Y 22.4754, Z -5.5000, A 0.000, B 0.000, C 0.000 }
gfCNCPoint4[1048] = {X 16.4765, Y 22.3119, Z -5.5000, A 0.000, B 0.000, C 0.000 }
gfCNCPoint4[1049] = {X 17.2351, Y 22.2007, Z -5.5000, A 0.000, B 0.000, C 0.000 }
gfCNCPoint4[1050] = {X 17.9718, Y 21.9883, Z -5.5000, A 0.000, B 0.000, C 0.000 }
gfCNCPoint4[1051] = {X 18.0837, Y 21.4828, Z -5.5000, A 0.000, B 0.000, C 0.000 }
gfCNCPoint4[1052] = {X 18.0305, Y 20.9677, Z -5.5000, A 0.000, B 0.000, C 0.000 }
gfCNCPoint4[1053] = {X 17.8175, Y 20.4957, Z -5.5000, A 0.000, B 0.000, C 0.000 }
gfCNCPoint4[1054] = {X 17.4665, Y 20.1150, Z -5.5000, A 0.000, B 0.000, C 0.000 }
gfCNCPoint4[1055] = {X 16.4756, Y 19.5310, Z -5.5000, A 0.000, B 0.000, C 0.000 }
gfCNCPoint4[1056] = {X 15.3891, Y 19.1536, Z -5.5000, A 0.000, B 0.000, C 0.000 }
gfCNCPoint4[1057] = {X 14.0143, Y 18.9291, Z -5.5000, A 0.000, B 0.000, C 0.000 }
gfCNCPoint4[1058] = {X 12.6225, Y 18.8734, Z -5.5000, A 0.000, B 0.000, C 0.000 }
gfCNCPoint4[1059] = {X 11.2342, Y 18.9873, Z -5.5000, A 0.000, B 0.000, C 0.000 }
gfCNCPoint4[1060] = {X 10.5417, Y 19.0961, Z -5.5000, A 0.000, B 0.000, C 0.000 }
gfCNCPoint4[1061] = {X 9.5229, Y 19.3345, Z -5.5000, A 0.000, B 0.000, C 0.000 }
gfCNCPoint4[1062] = {X 8.5386, Y 19.6897, Z -5.5000, A 0.000, B 0.000, C 0.000 }
gfCNCPoint4[1063] = {X 7.6024, Y 20.1570, Z -5.5000, A 0.000, B 0.000, C 0.000 }
gfCNCPoint4[1064] = {X 7.5898, Y 20.3183, Z -5.5000, A 0.000, B 0.000, C 0.000 }
gfCNCPoint4[1065] = {X 7.4462, Y 21.0539, Z -5.5000, A 0.000, B 0.000, C 0.000 }
gfCNCPoint4[1066] = {X 7.1679, Y 21.7499, Z -5.5000, A 0.000, B 0.000, C 0.000 }
gfCNCPoint4[1067] = {X 6.7646, Y 22.3816, Z -5.5000, A 0.000, B 0.000, C 0.000 }
gfCNCPoint4[1068] = {X 6.2506, Y 22.9271, Z -5.5000, A 0.000, B 0.000, C 0.000 }
gfCNCPoint4[1069] = {X 6.2084, Y 22.9637, Z -5.5000, A 0.000, B 0.000, C 0.000 }
gfCNCPoint4[1070] = {X 6.1658, Y 22.9996, Z -5.5000, A 0.000, B 0.000, C 0.000 }
gfCNCPoint4[1071] = {X 6.1508, Y 23.0919, Z -5.5000, A 0.000, B 0.000, C 0.000 }
gfCNCPoint4[1072] = {X 6.2332, Y 23.0790, Z -5.5000, A 0.000, B 0.000, C 0.000 }
gfCNCPoint4[1073] = {X 6.3155, Y 23.0663, Z -5.5000, A 0.000, B 0.000, C 0.000 }
gfCNCPoint4[1074] = {X 8.4230, Y 22.8024, Z -5.5000, A 0.000, B 0.000, C 0.000 }
gfCNCPoint4[1075] = {X 10.5417, Y 22.6545, Z -5.5000, A 0.000, B 0.000, C 0.000 }
gfCNCPoint4[1076] = {X 11.1758, Y 22.6294, Z -5.5000, A 0.000, B 0.000, C 0.000 }
gfCNCPoint4[1077] = {X 11.8097, Y 22.6016, Z -5.5000, A 0.000, B 0.000, C 0.000 }
gfCNCPoint4[1078] = {X 11.7176, Y 20.6037, Z -5.5000, A 0.000, B 0.000, C 0.000 }
gfCNCPoint4[1079] = {X 11.7176, Y 20.6037, Z -2.5000, A 0.000, B 0.000, C 0.000 }
gfCNCPoint4[1080] = {X 11.7176, Y 20.6037, Z 11.0000, A 0.000, B 0.000, C 0.000 }
gfCNCPoint4[1081] = {X 11.7091, Y 37.8766, Z 11.0000, A 0.000, B 0.000, C 0.000 }
gfCNCPoint4[1082] = {X 11.7091, Y 37.8766, Z -1.6667, A 0.000, B 0.000, C 0.000 }
gfCNCPoint4[1083] = {X 12.5146, Y 37.9488, Z -1.8834, A 0.000, B 0.000, C 0.000 }
gfCNCPoint4[1084] = {X 14.1652, Y 37.8338, Z -2.3267, A 0.000, B 0.000, C 0.000 }
gfCNCPoint4[1085] = {X 15.7768, Y 37.4590, Z -2.7701, A 0.000, B 0.000, C 0.000 }
gfCNCPoint4[1086] = {X 16.5095, Y 37.1631, Z -2.9818, A 0.000, B 0.000, C 0.000 }
gfCNCPoint4[1087] = {X 17.3401, Y 36.8276, Z -3.2218, A 0.000, B 0.000, C 0.000 }
gfCNCPoint4[1088] = {X 18.2944, Y 36.3171, Z -3.5118, A 0.000, B 0.000, C 0.000 }
gfCNCPoint4[1089] = {X 19.0345, Y 35.8123, Z -3.7519, A 0.000, B 0.000, C 0.000 }
gfCNCPoint4[1090] = {X 19.0577, Y 35.2982, Z -3.8898, A 0.000, B 0.000, C 0.000 }
gfCNCPoint4[1091] = {X 19.2189, Y 34.6356, Z -4.0725, A 0.000, B 0.000, C 0.000 }
gfCNCPoint4[1092] = {X 19.4344, Y 34.1683, Z -4.2104, A 0.000, B 0.000, C 0.000 }
gfCNCPoint4[1093] = {X 18.2011, Y 34.4166, Z -4.5475, A 0.000, B 0.000, C 0.000 }
gfCNCPoint4[1094] = {X 17.3655, Y 34.5301, Z -4.7734, A 0.000, B 0.000, C 0.000 }
gfCNCPoint4[1095] = {X 16.1106, Y 34.6199, Z -5.1105, A 0.000, B 0.000, C 0.000 }
gfCNCPoint4[1096] = {X 15.3859, Y 34.6737, Z -5.3053, A 0.000, B 0.000, C 0.000 }
gfCNCPoint4[1097] = {X 14.6609, Y 34.7232, Z -5.5000, A 0.000, B 0.000, C 0.000 }
gfCNCPoint4[1098] = {X 12.2607, Y 34.8758, Z -5.5000, A 0.000, B 0.000, C 0.000 }
gfCNCPoint4[1099] = {X 9.8592, Y 35.0055, Z -5.5000, A 0.000, B 0.000, C 0.000 }
gfCNCPoint4[1100] = {X 8.7537, Y 35.0956, Z -5.5000, A 0.000, B 0.000, C 0.000 }
gfCNCPoint4[1101] = {X 7.6655, Y 35.3095, Z -5.5000, A 0.000, B 0.000, C 0.000 }
gfCNCPoint4[1102] = {X 7.6559, Y 35.3712, Z -5.5000, A 0.000, B 0.000, C 0.000 }
gfCNCPoint4[1103] = {X 7.6526, Y 35.4335, Z -5.5000, A 0.000, B 0.000, C 0.000 }
gfCNCPoint4[1104] = {X 7.7533, Y 36.0261, Z -5.5000, A 0.000, B 0.000, C 0.000 }
gfCNCPoint4[1105] = {X 8.0476, Y 36.5502, Z -5.5000, A 0.000, B 0.000, C 0.000 }
gfCNCPoint4[1106] = {X 8.5013, Y 36.9445, Z -5.5000, A 0.000, B 0.000, C 0.000 }
gfCNCPoint4[1107] = {X 9.2758, Y 37.3370, Z -5.5000, A 0.000, B 0.000, C 0.000 }
gfCNCPoint4[1108] = {X 10.1000, Y 37.6096, Z -5.5000, A 0.000, B 0.000, C 0.000 }
gfCNCPoint4[1109] = {X 11.3840, Y 37.8458, Z -5.5000, A 0.000, B 0.000, C 0.000 }
gfCNCPoint4[1110] = {X 12.6875, Y 37.9190, Z -5.5000, A 0.000, B 0.000, C 0.000 }
gfCNCPoint4[1111] = {X 13.9899, Y 37.8283, Z -5.5000, A 0.000, B 0.000, C 0.000 }
gfCNCPoint4[1112] = {X 15.2706, Y 37.5750, Z -5.5000, A 0.000, B 0.000, C 0.000 }
gfCNCPoint4[1113] = {X 16.5095, Y 37.1631, Z -5.5000, A 0.000, B 0.000, C 0.000 }
gfCNCPoint4[1114] = {X 17.8083, Y 36.5555, Z -5.5000, A 0.000, B 0.000, C 0.000 }
gfCNCPoint4[1115] = {X 19.0345, Y 35.8123, Z -5.5000, A 0.000, B 0.000, C 0.000 }
gfCNCPoint4[1116] = {X 19.1547, Y 34.9709, Z -5.5000, A 0.000, B 0.000, C 0.000 }
gfCNCPoint4[1117] = {X 19.4344, Y 34.1683, Z -5.5000, A 0.000, B 0.000, C 0.000 }
gfCNCPoint4[1118] = {X 17.7797, Y 34.4470, Z -5.5000, A 0.000, B 0.000, C 0.000 }
gfCNCPoint4[1119] = {X 16.1106, Y 34.6199, Z -5.5000, A 0.000, B 0.000, C 0.000 }
gfCNCPoint4[1120] = {X 15.3858, Y 34.6726, Z -5.5000, A 0.000, B 0.000, C 0.000 }
gfCNCPoint4[1121] = {X 14.6609, Y 34.7232, Z -5.5000, A 0.000, B 0.000, C 0.000 }
gfCNCPoint4[1122] = {X 18.6547, Y 34.7194, Z -5.5000, A 0.000, B 0.000, C 0.000 }
gfCNCPoint4[1123] = {X 14.6554, Y 34.6434, Z -5.5000, A 0.000, B 0.000, C 0.000 }
gfCNCPoint4[1124] = {X 12.2589, Y 34.7958, Z -5.5000, A 0.000, B 0.000, C 0.000 }
gfCNCPoint4[1125] = {X 9.8611, Y 34.9255, Z -5.5000, A 0.000, B 0.000, C 0.000 }
gfCNCPoint4[1126] = {X 8.7209, Y 35.0194, Z -5.5000, A 0.000, B 0.000, C 0.000 }
gfCNCPoint4[1127] = {X 7.5992, Y 35.2440, Z -5.5000, A 0.000, B 0.000, C 0.000 }
gfCNCPoint4[1128] = {X 7.5794, Y 35.3377, Z -5.5000, A 0.000, B 0.000, C 0.000 }
gfCNCPoint4[1129] = {X 7.5726, Y 35.4332, Z -5.5000, A 0.000, B 0.000, C 0.000 }
gfCNCPoint4[1130] = {X 7.6778, Y 36.0528, Z -5.5000, A 0.000, B 0.000, C 0.000 }
gfCNCPoint4[1131] = {X 7.9856, Y 36.6007, Z -5.5000, A 0.000, B 0.000, C 0.000 }
gfCNCPoint4[1132] = {X 8.4600, Y 37.0130, Z -5.5000, A 0.000, B 0.000, C 0.000 }
gfCNCPoint4[1133] = {X 9.2450, Y 37.4108, Z -5.5000, A 0.000, B 0.000, C 0.000 }
gfCNCPoint4[1134] = {X 10.0806, Y 37.6873, Z -5.5000, A 0.000, B 0.000, C 0.000 }
gfCNCPoint4[1135] = {X 11.3745, Y 37.9252, Z -5.5000, A 0.000, B 0.000, C 0.000 }
gfCNCPoint4[1136] = {X 12.6880, Y 37.9990, Z -5.5000, A 0.000, B 0.000, C 0.000 }
gfCNCPoint4[1137] = {X 14.0004, Y 37.9076, Z -5.5000, A 0.000, B 0.000, C 0.000 }
gfCNCPoint4[1138] = {X 15.2910, Y 37.6523, Z -5.5000, A 0.000, B 0.000, C 0.000 }
gfCNCPoint4[1139] = {X 16.5394, Y 37.2373, Z -5.5000, A 0.000, B 0.000, C 0.000 }
gfCNCPoint4[1140] = {X 17.8637, Y 36.6166, Z -5.5000, A 0.000, B 0.000, C 0.000 }
gfCNCPoint4[1141] = {X 19.1128, Y 35.8557, Z -5.5000, A 0.000, B 0.000, C 0.000 }
gfCNCPoint4[1142] = {X 19.2471, Y 34.9313, Z -5.5000, A 0.000, B 0.000, C 0.000 }
gfCNCPoint4[1143] = {X 19.5769, Y 34.0574, Z -5.5000, A 0.000, B 0.000, C 0.000 }
gfCNCPoint4[1144] = {X 17.8489, Y 34.3567, Z -5.5000, A 0.000, B 0.000, C 0.000 }
gfCNCPoint4[1145] = {X 16.1048, Y 34.5401, Z -5.5000, A 0.000, B 0.000, C 0.000 }
gfCNCPoint4[1146] = {X 15.3802, Y 34.5928, Z -5.5000, A 0.000, B 0.000, C 0.000 }
gfCNCPoint4[1147] = {X 14.6554, Y 34.6434, Z -5.5000, A 0.000, B 0.000, C 0.000 }
gfCNCPoint4[1148] = {X 10.7037, Y 35.2631, Z -5.5000, A 0.000, B 0.000, C 0.000 }
gfCNCPoint4[1149] = {X 18.6492, Y 34.6396, Z -5.5000, A 0.000, B 0.000, C 0.000 }
gfCNCPoint4[1150] = {X 14.6500, Y 34.5636, Z -5.5000, A 0.000, B 0.000, C 0.000 }
gfCNCPoint4[1151] = {X 12.2547, Y 34.7160, Z -5.5000, A 0.000, B 0.000, C 0.000 }
gfCNCPoint4[1152] = {X 9.8581, Y 34.8455, Z -5.5000, A 0.000, B 0.000, C 0.000 }
gfCNCPoint4[1153] = {X 8.6874, Y 34.9434, Z -5.5000, A 0.000, B 0.000, C 0.000 }
gfCNCPoint4[1154] = {X 7.5362, Y 35.1779, Z -5.5000, A 0.000, B 0.000, C 0.000 }
gfCNCPoint4[1155] = {X 7.5038, Y 35.3036, Z -5.5000, A 0.000, B 0.000, C 0.000 }
gfCNCPoint4[1156] = {X 7.4926, Y 35.4329, Z -5.5000, A 0.000, B 0.000, C 0.000 }
gfCNCPoint4[1157] = {X 7.6024, Y 36.0795, Z -5.5000, A 0.000, B 0.000, C 0.000 }
gfCNCPoint4[1158] = {X 7.9236, Y 36.6512, Z -5.5000, A 0.000, B 0.000, C 0.000 }
gfCNCPoint4[1159] = {X 8.4186, Y 37.0815, Z -5.5000, A 0.000, B 0.000, C 0.000 }
gfCNCPoint4[1160] = {X 9.2143, Y 37.4847, Z -5.5000, A 0.000, B 0.000, C 0.000 }
gfCNCPoint4[1161] = {X 10.0612, Y 37.7649, Z -5.5000, A 0.000, B 0.000, C 0.000 }
gfCNCPoint4[1162] = {X 11.3650, Y 38.0046, Z -5.5000, A 0.000, B 0.000, C 0.000 }
gfCNCPoint4[1163] = {X 12.6886, Y 38.0790, Z -5.5000, A 0.000, B 0.000, C 0.000 }
gfCNCPoint4[1164] = {X 14.0110, Y 37.9869, Z -5.5000, A 0.000, B 0.000, C 0.000 }
gfCNCPoint4[1165] = {X 15.3115, Y 37.7297, Z -5.5000, A 0.000, B 0.000, C 0.000 }
gfCNCPoint4[1166] = {X 16.5694, Y 37.3114, Z -5.5000, A 0.000, B 0.000, C 0.000 }
gfCNCPoint4[1167] = {X 17.9195, Y 36.6775, Z -5.5000, A 0.000, B 0.000, C 0.000 }
gfCNCPoint4[1168] = {X 19.1915, Y 35.8986, Z -5.5000, A 0.000, B 0.000, C 0.000 }
gfCNCPoint4[1169] = {X 19.2642, Y 35.2209, Z -5.5000, A 0.000, B 0.000, C 0.000 }
gfCNCPoint4[1170] = {X 19.4447, Y 34.5636, Z -5.5000, A 0.000, B 0.000, C 0.000 }
gfCNCPoint4[1171] = {X 19.7281, Y 33.9438, Z -5.5000, A 0.000, B 0.000, C 0.000 }
gfCNCPoint4[1172] = {X 17.9226, Y 34.2656, Z -5.5000, A 0.000, B 0.000, C 0.000 }
gfCNCPoint4[1173] = {X 16.0990, Y 34.4603, Z -5.5000, A 0.000, B 0.000, C 0.000 }
gfCNCPoint4[1174] = {X 15.3746, Y 34.5130, Z -5.5000, A 0.000, B 0.000, C 0.000 }
gfCNCPoint4[1175] = {X 14.6500, Y 34.5636, Z -5.5000, A 0.000, B 0.000, C 0.000 }
gfCNCPoint4[1176] = {X 10.6982, Y 35.1833, Z -5.5000, A 0.000, B 0.000, C 0.000 }
gfCNCPoint4[1177] = {X 18.6438, Y 34.5597, Z -5.5000, A 0.000, B 0.000, C 0.000 }
gfCNCPoint4[1178] = {X 14.6445, Y 34.4838, Z -5.5000, A 0.000, B 0.000, C 0.000 }
gfCNCPoint4[1179] = {X 12.2505, Y 34.6361, Z -5.5000, A 0.000, B 0.000, C 0.000 }
gfCNCPoint4[1180] = {X 9.8551, Y 34.7656, Z -5.5000, A 0.000, B 0.000, C 0.000 }
gfCNCPoint4[1181] = {X 8.6552, Y 34.8672, Z -5.5000, A 0.000, B 0.000, C 0.000 }
gfCNCPoint4[1182] = {X 7.4759, Y 35.1112, Z -5.5000, A 0.000, B 0.000, C 0.000 }
gfCNCPoint4[1183] = {X 7.4288, Y 35.2689, Z -5.5000, A 0.000, B 0.000, C 0.000 }
gfCNCPoint4[1184] = {X 7.4126, Y 35.4326, Z -5.5000, A 0.000, B 0.000, C 0.000 }
gfCNCPoint4[1185] = {X 7.5270, Y 36.1061, Z -5.5000, A 0.000, B 0.000, C 0.000 }
gfCNCPoint4[1186] = {X 7.8616, Y 36.7018, Z -5.5000, A 0.000, B 0.000, C 0.000 }
gfCNCPoint4[1187] = {X 8.3772, Y 37.1499, Z -5.5000, A 0.000, B 0.000, C 0.000 }
gfCNCPoint4[1188] = {X 9.1836, Y 37.5586, Z -5.5000, A 0.000, B 0.000, C 0.000 }
gfCNCPoint4[1189] = {X 10.0418, Y 37.8425, Z -5.5000, A 0.000, B 0.000, C 0.000 }
gfCNCPoint4[1190] = {X 11.3555, Y 38.0841, Z -5.5000, A 0.000, B 0.000, C 0.000 }
gfCNCPoint4[1191] = {X 12.6891, Y 38.1590, Z -5.5000, A 0.000, B 0.000, C 0.000 }
gfCNCPoint4[1192] = {X 14.0216, Y 38.0662, Z -5.5000, A 0.000, B 0.000, C 0.000 }
gfCNCPoint4[1193] = {X 15.3319, Y 37.8070, Z -5.5000, A 0.000, B 0.000, C 0.000 }
gfCNCPoint4[1194] = {X 16.5994, Y 37.3856, Z -5.5000, A 0.000, B 0.000, C 0.000 }
gfCNCPoint4[1195] = {X 17.9754, Y 36.7382, Z -5.5000, A 0.000, B 0.000, C 0.000 }
gfCNCPoint4[1196] = {X 19.2706, Y 35.9411, Z -5.5000, A 0.000, B 0.000, C 0.000 }
gfCNCPoint4[1197] = {X 19.3492, Y 35.2030, Z -5.5000, A 0.000, B 0.000, C 0.000 }
gfCNCPoint4[1198] = {X 19.5578, Y 34.4906, Z -5.5000, A 0.000, B 0.000, C 0.000 }
gfCNCPoint4[1199] = {X 19.8896, Y 33.8266, Z -5.5000, A 0.000, B 0.000, C 0.000 }
gfCNCPoint4[1200] = {X 18.0016, Y 34.1734, Z -5.5000, A 0.000, B 0.000, C 0.000 }
gfCNCPoint4[1201] = {X 16.0932, Y 34.3805, Z -5.5000, A 0.000, B 0.000, C 0.000 }
gfCNCPoint4[1202] = {X 15.3689, Y 34.4332, Z -5.5000, A 0.000, B 0.000, C 0.000 }
gfCNCPoint4[1203] = {X 14.6445, Y 34.4838, Z -5.5000, A 0.000, B 0.000, C 0.000 }
gfCNCPoint4[1204] = {X 10.6928, Y 35.1035, Z -5.5000, A 0.000, B 0.000, C 0.000 }
gfCNCPoint4[1205] = {X 18.6383, Y 34.4799, Z -5.5000, A 0.000, B 0.000, C 0.000 }
gfCNCPoint4[1206] = {X 14.6390, Y 34.4040, Z -5.5000, A 0.000, B 0.000, C 0.000 }
gfCNCPoint4[1207] = {X 12.2463, Y 34.5562, Z -5.5000, A 0.000, B 0.000, C 0.000 }
gfCNCPoint4[1208] = {X 9.8522, Y 34.6856, Z -5.5000, A 0.000, B 0.000, C 0.000 }
gfCNCPoint4[1209] = {X 8.6240, Y 34.7909, Z -5.5000, A 0.000, B 0.000, C 0.000 }
gfCNCPoint4[1210] = {X 7.4177, Y 35.0441, Z -5.5000, A 0.000, B 0.000, C 0.000 }
gfCNCPoint4[1211] = {X 7.3544, Y 35.2337, Z -5.5000, A 0.000, B 0.000, C 0.000 }
gfCNCPoint4[1212] = {X 7.3326, Y 35.4324, Z -5.5000, A 0.000, B 0.000, C 0.000 }
gfCNCPoint4[1213] = {X 7.3993, Y 35.9622, Z -5.5000, A 0.000, B 0.000, C 0.000 }
gfCNCPoint4[1214] = {X 7.5989, Y 36.4575, Z -5.5000, A 0.000, B 0.000, C 0.000 }
gfCNCPoint4[1215] = {X 7.9181, Y 36.8857, Z -5.5000, A 0.000, B 0.000, C 0.000 }
gfCNCPoint4[1216] = {X 8.3358, Y 37.2184, Z -5.5000, A 0.000, B 0.000, C 0.000 }
gfCNCPoint4[1217] = {X 9.1528, Y 37.6324, Z -5.5000, A 0.000, B 0.000, C 0.000 }
gfCNCPoint4[1218] = {X 10.0225, Y 37.9201, Z -5.5000, A 0.000, B 0.000, C 0.000 }
gfCNCPoint4[1219] = {X 11.3460, Y 38.1635, Z -5.5000, A 0.000, B 0.000, C 0.000 }
gfCNCPoint4[1220] = {X 12.6896, Y 38.2390, Z -5.5000, A 0.000, B 0.000, C 0.000 }
gfCNCPoint4[1221] = {X 14.0321, Y 38.1455, Z -5.5000, A 0.000, B 0.000, C 0.000 }
gfCNCPoint4[1222] = {X 15.3523, Y 37.8844, Z -5.5000, A 0.000, B 0.000, C 0.000 }
gfCNCPoint4[1223] = {X 16.6293, Y 37.4598, Z -5.5000, A 0.000, B 0.000, C 0.000 }
gfCNCPoint4[1224] = {X 18.0316, Y 36.7987, Z -5.5000, A 0.000, B 0.000, C 0.000 }
gfCNCPoint4[1225] = {X 19.3501, Y 35.9832, Z -5.5000, A 0.000, B 0.000, C 0.000 }
gfCNCPoint4[1226] = {X 19.4352, Y 35.1815, Z -5.5000, A 0.000, B 0.000, C 0.000 }
gfCNCPoint4[1227] = {X 19.6763, Y 34.4121, Z -5.5000, A 0.000, B 0.000, C 0.000 }
gfCNCPoint4[1228] = {X 20.0640, Y 33.7052, Z -5.5000, A 0.000, B 0.000, C 0.000 }
